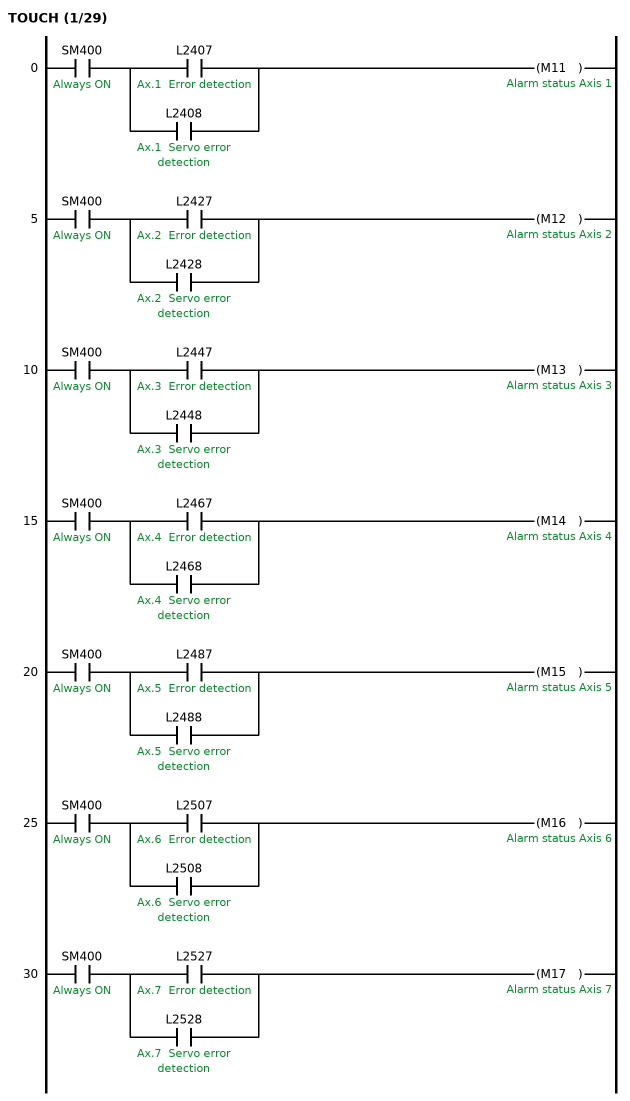
[picture p48: ladder of TOUCH, rungs at steps 0 to 30]
0     LD      SM400  ; Always ON
      LD      L2407  ; Ax.1  Error detection
      OR      L2408  ; Ax.1  Servo error detection
      ANB
      OUT     M11  ; Alarm status Axis 1
5     LD      SM400  ; Always ON
      LD      L2427  ; Ax.2  Error detection
      OR      L2428  ; Ax.2  Servo error detection
      ANB
      OUT     M12  ; Alarm status Axis 2
10    LD      SM400  ; Always ON
      LD      L2447  ; Ax.3  Error detection
      OR      L2448  ; Ax.3  Servo error detection
      ANB
      OUT     M13  ; Alarm status Axis 3
15    LD      SM400  ; Always ON
      LD      L2467  ; Ax.4  Error detection
      OR      L2468  ; Ax.4  Servo error detection
      ANB
      OUT     M14  ; Alarm status Axis 4
20    LD      SM400  ; Always ON
      LD      L2487  ; Ax.5  Error detection
      OR      L2488  ; Ax.5  Servo error detection
      ANB
      OUT     M15  ; Alarm status Axis 5
25    LD      SM400  ; Always ON
      LD      L2507  ; Ax.6  Error detection
      OR      L2508  ; Ax.6  Servo error detection
      ANB
      OUT     M16  ; Alarm status Axis 6
30    LD      SM400  ; Always ON
      LD      L2527  ; Ax.7  Error detection
      OR      L2528  ; Ax.7  Servo error detection
      ANB
      OUT     M17  ; Alarm status Axis 7
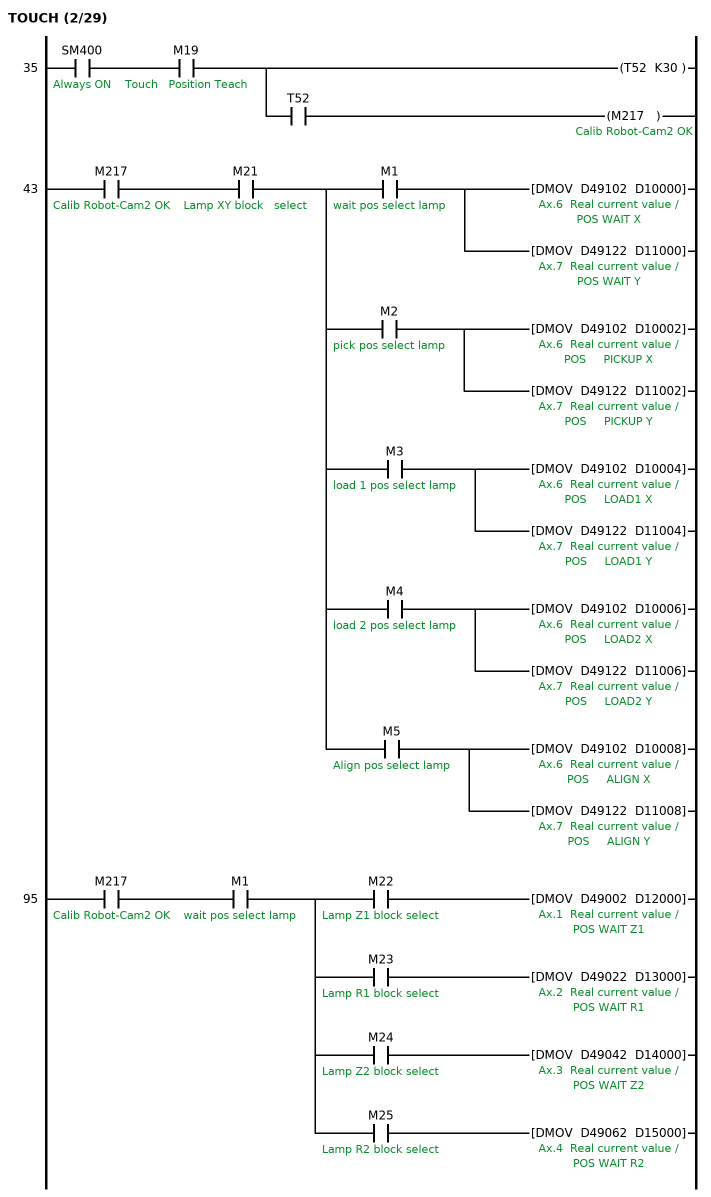
35    LD      SM400  ; Always ON
      AND     M19  ; Touch   Position Teach
      OUT     T52 K30
      AND     T52
      OUT     M217  ; Calib Robot-Cam2 OK
43    LD      M217  ; Calib Robot-Cam2 OK
      AND     M21  ; Lamp XY block   select
      MPS
      AND     M1  ; wait pos select lamp
      DMOV    D49102 D10000  ; Ax.6  Real current value / POS WAIT X
      DMOV    D49122 D11000  ; Ax.7  Real current value / POS WAIT Y
      MRD
      AND     M2  ; pick pos select lamp
      DMOV    D49102 D10002  ; POS     PICKUP X
      DMOV    D49122 D11002  ; POS     PICKUP Y
      MRD
      AND     M3  ; load 1 pos select lamp
      DMOV    D49102 D10004  ; POS     LOAD1 X
      DMOV    D49122 D11004  ; POS     LOAD1 Y
      MRD
      AND     M4  ; load 2 pos select lamp
      DMOV    D49102 D10006  ; POS     LOAD2 X
      DMOV    D49122 D11006  ; POS     LOAD2 Y
      MPP
      AND     M5  ; Align pos select lamp
      DMOV    D49102 D10008  ; POS     ALIGN X
      DMOV    D49122 D11008  ; POS     ALIGN Y
95    LD      M217  ; Calib Robot-Cam2 OK
      AND     M1  ; wait pos select lamp
      MPS
      AND     M22  ; Lamp Z1 block select
      DMOV    D49002 D12000  ; Ax.1  Real current value / POS WAIT Z1
      MRD
      AND     M23  ; Lamp R1 block select
      DMOV    D49022 D13000  ; Ax.2  Real current value / POS WAIT R1
      MRD
      AND     M24  ; Lamp Z2 block select
      DMOV    D49042 D14000  ; Ax.3  Real current value / POS WAIT Z2
      MPP
      AND     M25  ; Lamp R2 block select
      DMOV    D49062 D15000  ; Ax.4  Real current value / POS WAIT R2
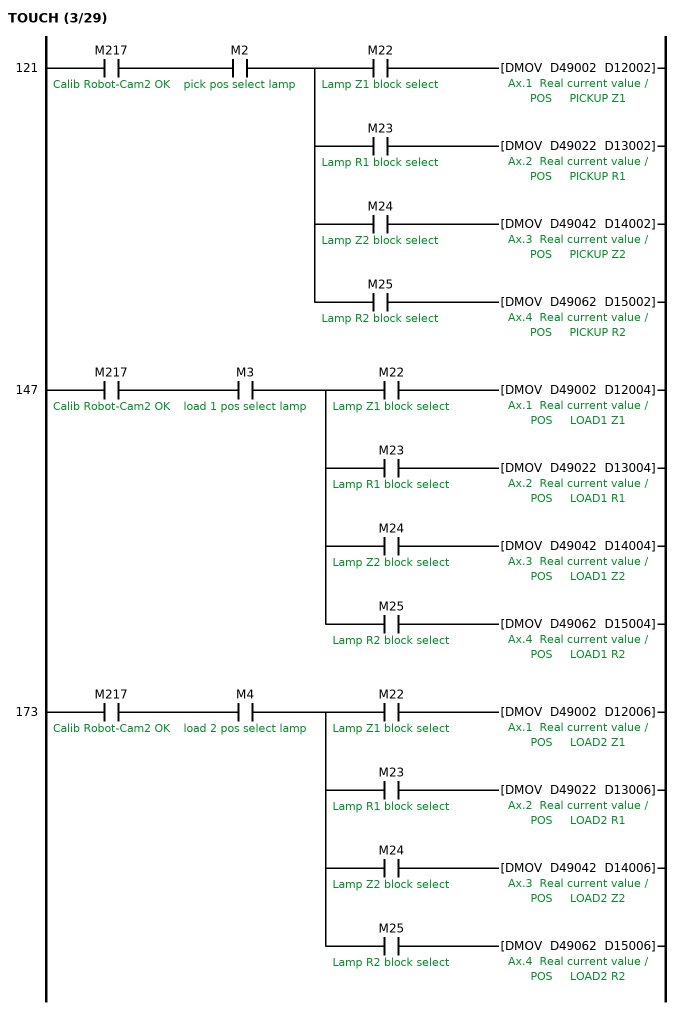
121   LD      M217  ; Calib Robot-Cam2 OK
      AND     M2  ; pick pos select lamp
      MPS
      AND     M22  ; Lamp Z1 block select
      DMOV    D49002 D12002  ; POS     PICKUP Z1
      MRD
      AND     M23  ; Lamp R1 block select
      DMOV    D49022 D13002  ; POS     PICKUP R1
      MRD
      AND     M24  ; Lamp Z2 block select
      DMOV    D49042 D14002  ; POS     PICKUP Z2
      MPP
      AND     M25  ; Lamp R2 block select
      DMOV    D49062 D15002  ; POS     PICKUP R2
147   LD      M217  ; Calib Robot-Cam2 OK
      AND     M3  ; load 1 pos select lamp
      MPS
      AND     M22  ; Lamp Z1 block select
      DMOV    D49002 D12004  ; POS     LOAD1 Z1
      MRD
      AND     M23  ; Lamp R1 block select
      DMOV    D49022 D13004  ; POS     LOAD1 R1
      MRD
      AND     M24  ; Lamp Z2 block select
      DMOV    D49042 D14004  ; POS     LOAD1 Z2
      MPP
      AND     M25  ; Lamp R2 block select
      DMOV    D49062 D15004  ; POS     LOAD1 R2
173   LD      M217  ; Calib Robot-Cam2 OK
      AND     M4  ; load 2 pos select lamp
      MPS
      AND     M22  ; Lamp Z1 block select
      DMOV    D49002 D12006  ; POS     LOAD2 Z1
      MRD
      AND     M23  ; Lamp R1 block select
      DMOV    D49022 D13006  ; POS     LOAD2 R1
      MRD
      AND     M24  ; Lamp Z2 block select
      DMOV    D49042 D14006  ; POS     LOAD2 Z2
      MPP
      AND     M25  ; Lamp R2 block select
      DMOV    D49062 D15006  ; POS     LOAD2 R2
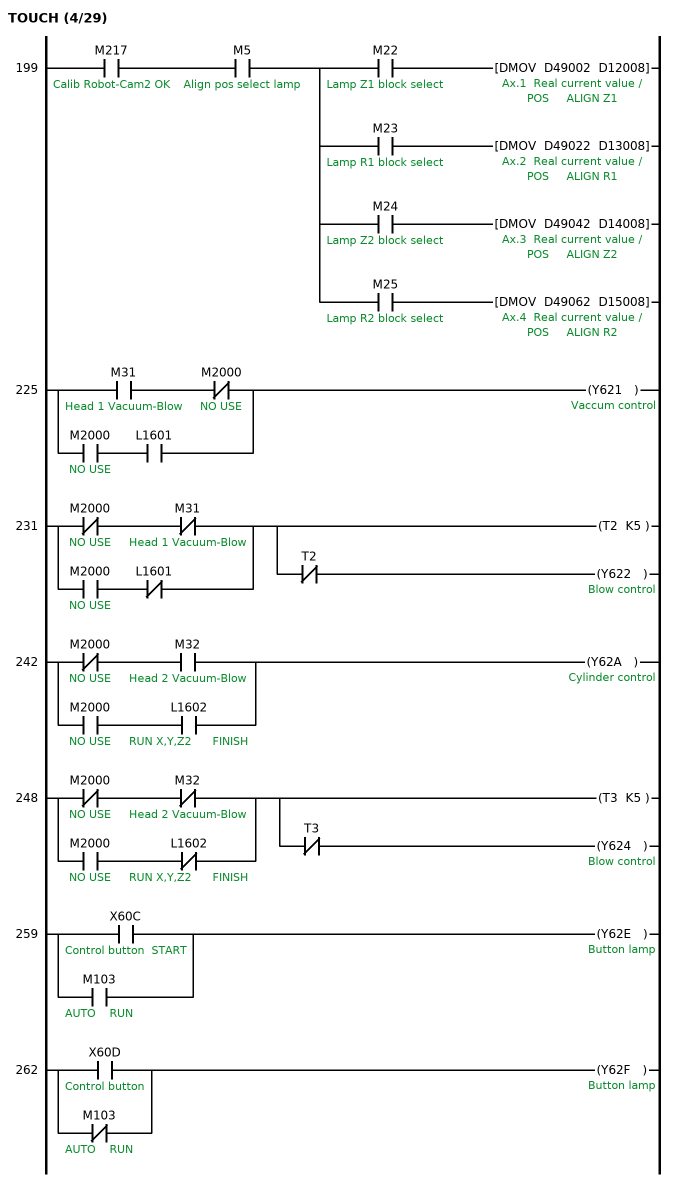
199   LD      M217  ; Calib Robot-Cam2 OK
      AND     M5  ; Align pos select lamp
      MPS
      AND     M22  ; Lamp Z1 block select
      DMOV    D49002 D12008  ; POS     ALIGN Z1
      MRD
      AND     M23  ; Lamp R1 block select
      DMOV    D49022 D13008  ; POS     ALIGN R1
      MRD
      AND     M24  ; Lamp Z2 block select
      DMOV    D49042 D14008  ; POS     ALIGN Z2
      MPP
      AND     M25  ; Lamp R2 block select
      DMOV    D49062 D15008  ; POS     ALIGN R2
225   LD      M31  ; Head 1 Vacuum-Blow
      ANI     M2000  ; NO USE
      LD      M2000  ; NO USE
      AND     L1601
      ORB
      OUT     Y621  ; Vaccum control
231   LDI     M2000  ; NO USE
      ANI     M31  ; Head 1 Vacuum-Blow
      LD      M2000  ; NO USE
      ANI     L1601
      ORB
      OUT     T2 K5
      ANI     T2
      OUT     Y622  ; Blow control
242   LDI     M2000  ; NO USE
      AND     M32  ; Head 2 Vacuum-Blow
      LD      M2000  ; NO USE
      AND     L1602  ; RUN X,Y,Z2      FINISH
      ORB
      OUT     Y62A  ; Cylinder control
248   LDI     M2000  ; NO USE
      ANI     M32  ; Head 2 Vacuum-Blow
      LD      M2000  ; NO USE
      ANI     L1602  ; RUN X,Y,Z2      FINISH
      ORB
      OUT     T3 K5
      ANI     T3
      OUT     Y624  ; Blow control
259   LD      X60C  ; Control button  START
      OR      M103  ; AUTO    RUN
      OUT     Y62E  ; Button lamp
262   LD      X60D  ; Control button
      ORI     M103  ; AUTO    RUN
      OUT     Y62F  ; Button lamp
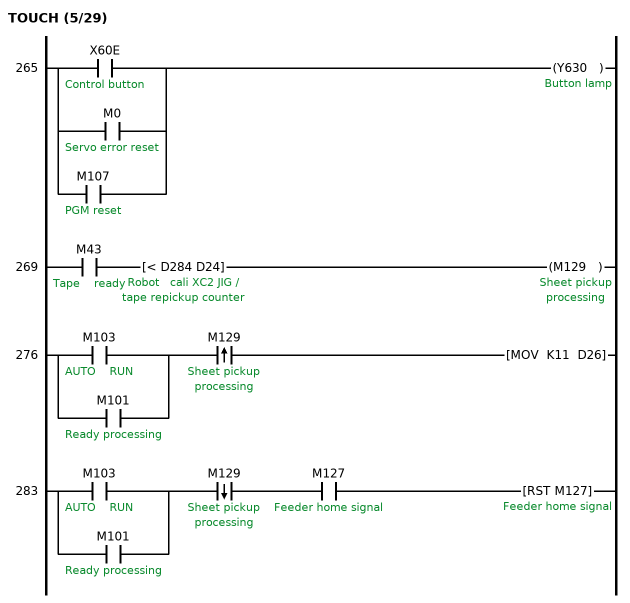
265   LD      X60E  ; Control button
      OR      M0  ; Servo error reset
      OR      M107  ; PGM reset
      OUT     Y630  ; Button lamp
269   LD      M43  ; Tape    ready
      AND<    D284 D24  ; Robot   cali XC2 JIG / tape repickup counter
      OUT     M129  ; Sheet pickup processing
276   LD      M103  ; AUTO    RUN
      OR      M101  ; Ready processing
      ANDP    M129  ; Sheet pickup processing
      MOV     K11 D26
283   LD      M103  ; AUTO    RUN
      OR      M101  ; Ready processing
      ANDF    M129  ; Sheet pickup processing
      AND     M127  ; Feeder home signal
      RST     M127  ; Feeder home signal
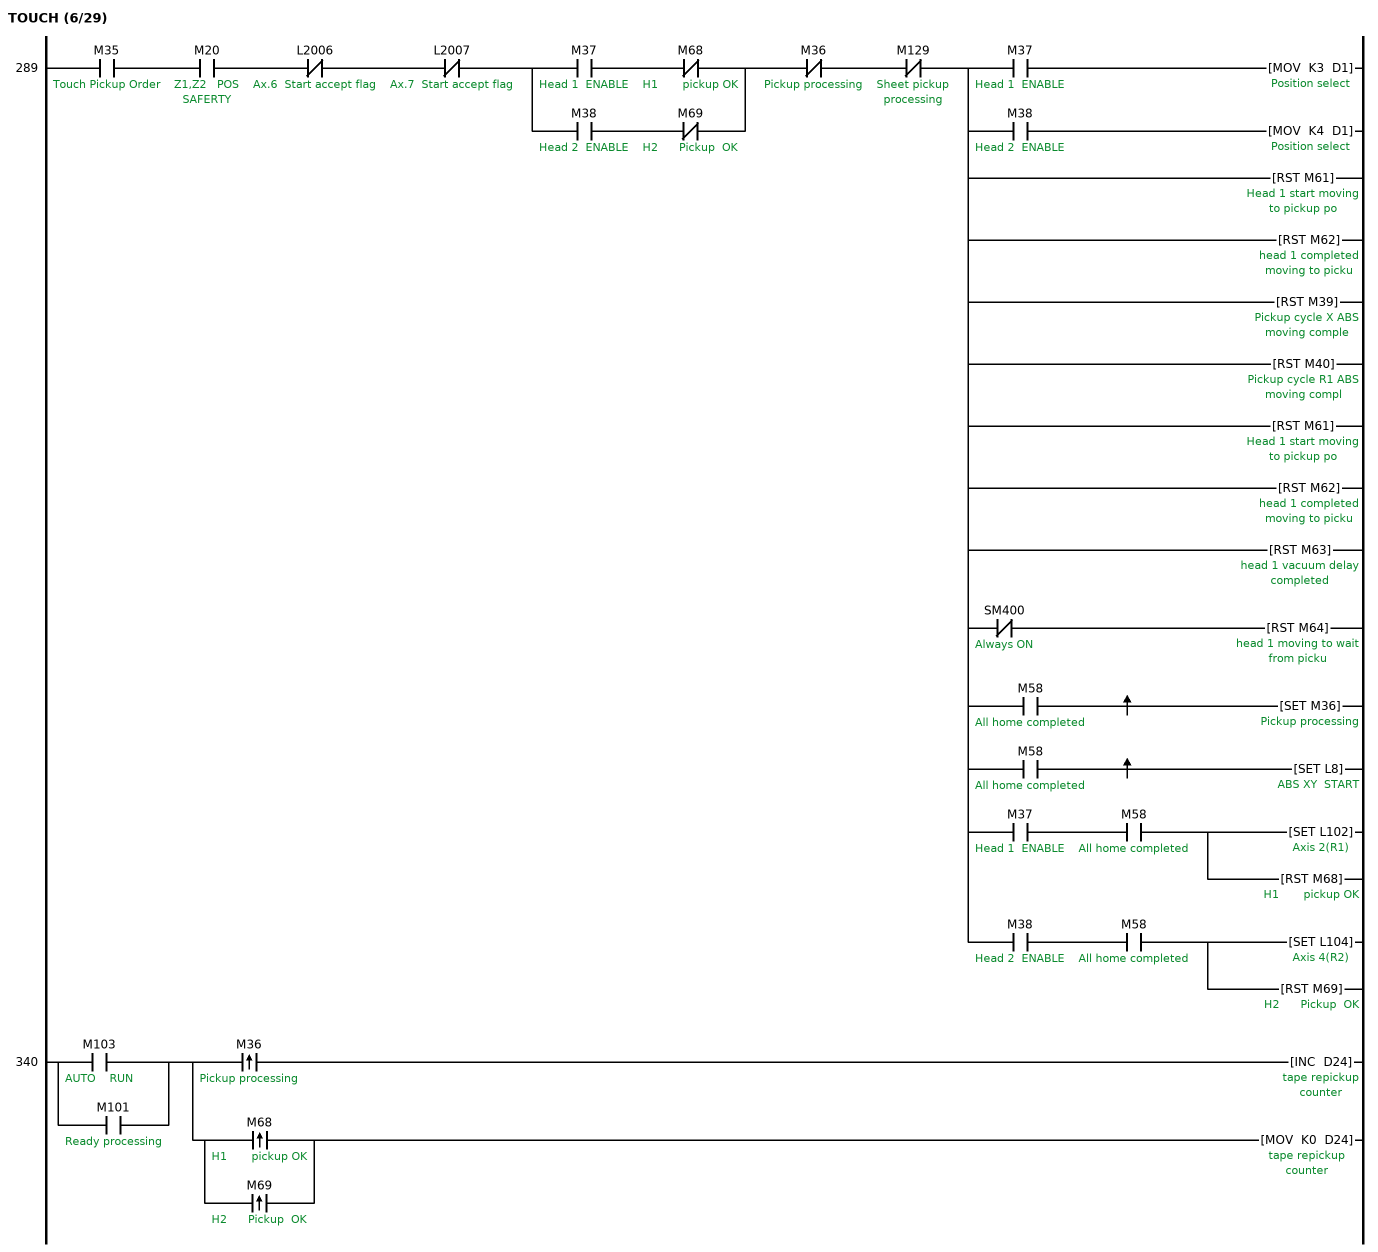
289   LD      M35  ; Touch Pickup Order
      AND     M20  ; Z1,Z2   POS     SAFERTY
      ANI     L2006  ; Ax.6  Start accept flag
      ANI     L2007  ; Ax.7  Start accept flag
      LD      M37  ; Head 1  ENABLE
      ANI     M68  ; H1       pickup OK
      LD      M38  ; Head 2  ENABLE
      ANI     M69  ; H2      Pickup  OK
      ORB
      ANB
      ANI     M36  ; Pickup processing
      ANI     M129  ; Sheet pickup processing
      MPS
      AND     M37  ; Head 1  ENABLE
      MOV     K3 D1  ; Position select
      MRD
      AND     M38  ; Head 2  ENABLE
      MOV     K4 D1
      MPP
      RST     M61  ; Head 1 start moving to pickup po
      RST     M62  ; head 1 completed moving to picku
      RST     M39  ; Pickup cycle X ABS moving comple
      RST     M40  ; Pickup cycle R1 ABS moving compl
      RST     M61  ; Head 1 start moving to pickup po
      RST     M62  ; head 1 completed moving to picku
      RST     M63  ; head 1 vacuum delay completed
      MPS
      ANI     SM400  ; Always ON
      RST     M64  ; head 1 moving to wait from picku
      MRD
      AND     M58  ; All home completed
      MEP
      SET     M36  ; Pickup processing
      MRD
      AND     M58  ; All home completed
      MEP
      SET     L8  ; ABS XY  START
      MRD
      AND     M37  ; Head 1  ENABLE
      AND     M58  ; All home completed
      SET     L102  ; Axis 2(R1)
      RST     M68  ; H1       pickup OK
      MPP
      AND     M38  ; Head 2  ENABLE
      AND     M58  ; All home completed
      SET     L104  ; Axis 4(R2)
      RST     M69  ; H2      Pickup  OK
340   LD      M103  ; AUTO    RUN
      OR      M101  ; Ready processing
      MPS
      ANDP    M36  ; Pickup processing
      INC     D24
      MPP
      LDP     M68  ; H1       pickup OK
      ORP     M69  ; H2      Pickup  OK
      ANB
      MOV     K0 D24
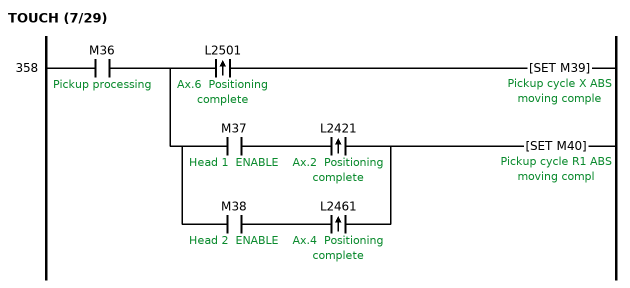
358   LD      M36  ; Pickup processing
      MPS
      ANDP    L2501  ; Ax.6  Positioning complete
      SET     M39  ; Pickup cycle X ABS moving comple
      MPP
      LD      M37  ; Head 1  ENABLE
      ANDP    L2421  ; Ax.2  Positioning complete
      LD      M38  ; Head 2  ENABLE
      ANDP    L2461  ; Ax.4  Positioning complete
      ORB
      ANB
      SET     M40  ; Pickup cycle R1 ABS moving compl
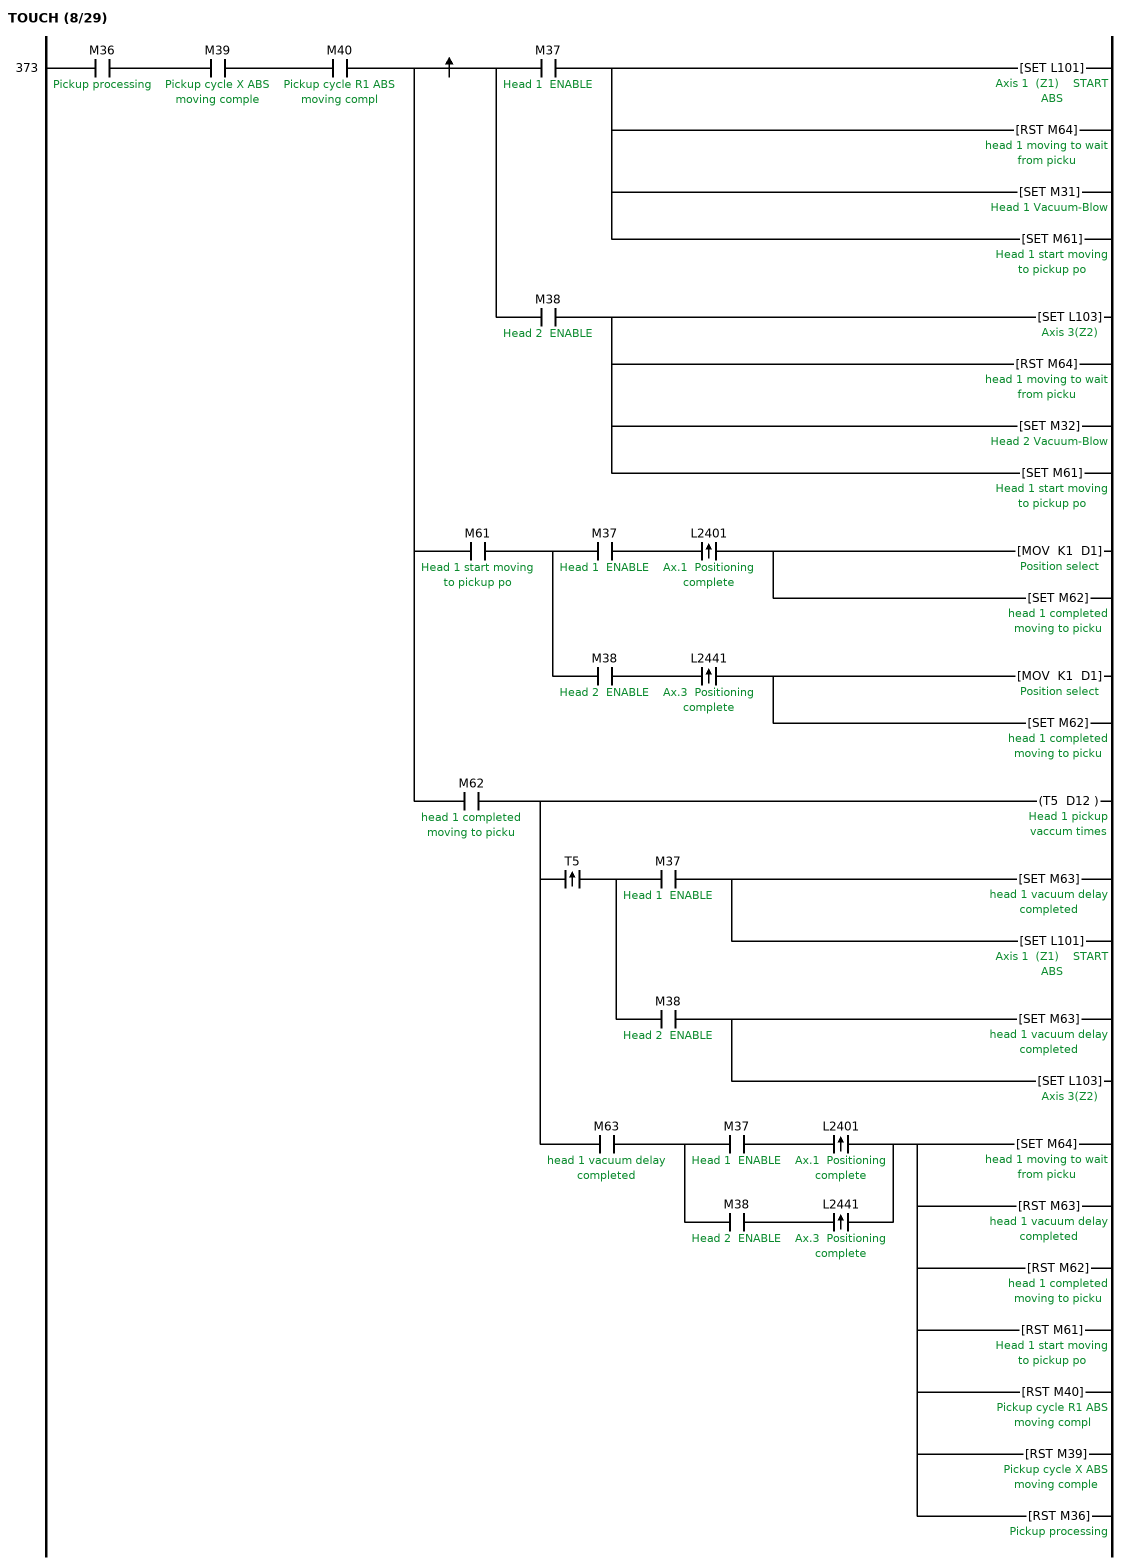
373   LD      M36  ; Pickup processing
      AND     M39  ; Pickup cycle X ABS moving comple
      AND     M40  ; Pickup cycle R1 ABS moving compl
      MPS
      MEP
      MPS
      AND     M37  ; Head 1  ENABLE
      SET     L101  ; Axis 1  (Z1)    START   ABS
      RST     M64  ; head 1 moving to wait from picku
      SET     M31  ; Head 1 Vacuum-Blow
      SET     M61  ; Head 1 start moving to pickup po
      MPP
      AND     M38  ; Head 2  ENABLE
      SET     L103  ; Axis 3(Z2)
      RST     M64  ; head 1 moving to wait from picku
      SET     M32  ; Head 2 Vacuum-Blow
      SET     M61  ; Head 1 start moving to pickup po
      MRD
      AND     M61  ; Head 1 start moving to pickup po
      MPS
      AND     M37  ; Head 1  ENABLE
      ANDP    L2401  ; Ax.1  Positioning complete
      MOV     K1 D1
      SET     M62  ; head 1 completed moving to picku
      MPP
      AND     M38  ; Head 2  ENABLE
      ANDP    L2441  ; Ax.3  Positioning complete
      MOV     K1 D1
      SET     M62  ; head 1 completed moving to picku
      MPP
      AND     M62  ; head 1 completed moving to picku
      OUT     T5 D12  ; Head 1 pickup vaccum times
      MPS
      ANDP    T5
      MPS
      AND     M37  ; Head 1  ENABLE
      SET     M63  ; head 1 vacuum delay completed
      SET     L101  ; Axis 1  (Z1)    START   ABS
      MPP
      AND     M38  ; Head 2  ENABLE
      SET     M63  ; head 1 vacuum delay completed
      SET     L103  ; Axis 3(Z2)
      MPP
      AND     M63  ; head 1 vacuum delay completed
      LD      M37  ; Head 1  ENABLE
      ANDP    L2401  ; Ax.1  Positioning complete
      LD      M38  ; Head 2  ENABLE
      ANDP    L2441  ; Ax.3  Positioning complete
      ORB
      ANB
      SET     M64  ; head 1 moving to wait from picku
      RST     M63  ; head 1 vacuum delay completed
      RST     M62  ; head 1 completed moving to picku
      RST     M61  ; Head 1 start moving to pickup po
      RST     M40  ; Pickup cycle R1 ABS moving compl
      RST     M39  ; Pickup cycle X ABS moving comple
      RST     M36  ; Pickup processing
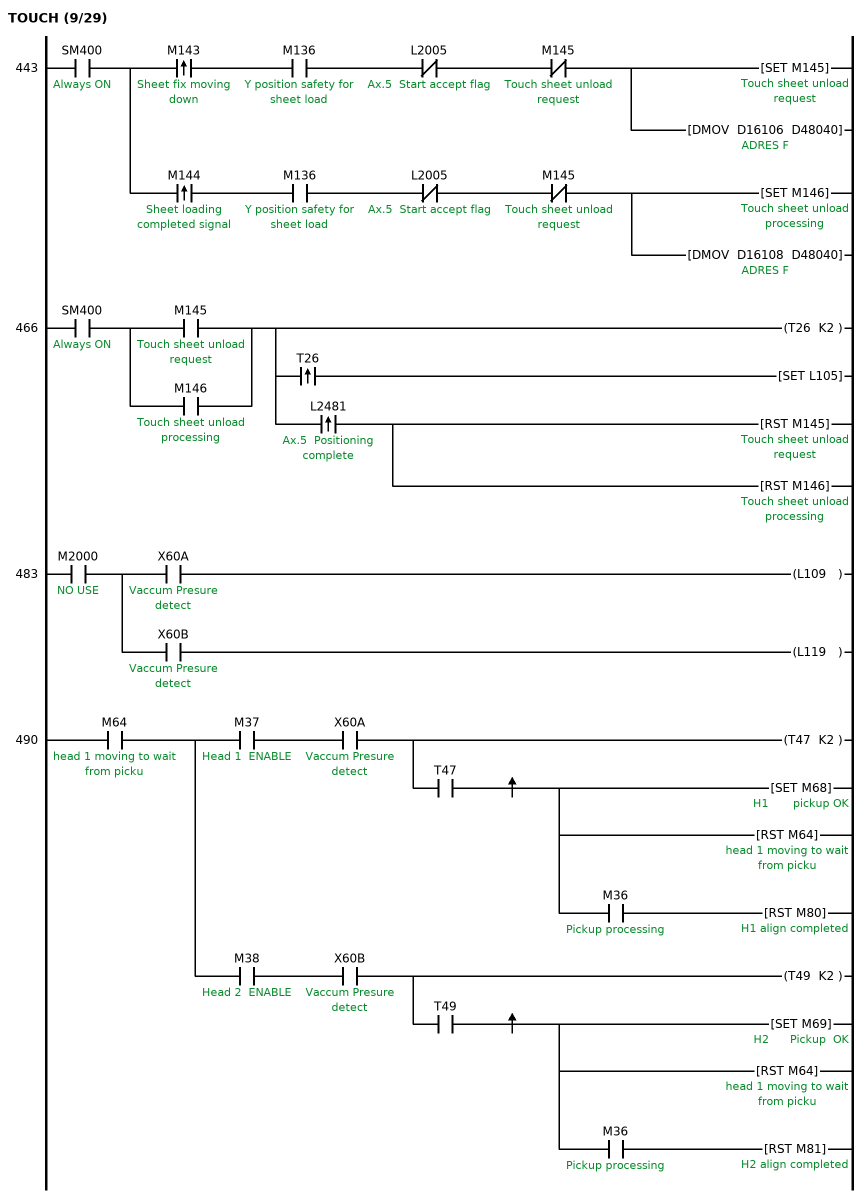
443   LD      SM400  ; Always ON
      MPS
      ANDP    M143  ; Sheet fix moving down
      AND     M136  ; Y position safety for sheet load
      ANI     L2005  ; Ax.5  Start accept flag
      ANI     M145  ; Touch sheet unload request
      SET     M145  ; Touch sheet unload request
      DMOV    D16106 D48040  ; ADRES F
      MPP
      ANDP    M144  ; Sheet loading completed signal
      AND     M136  ; Y position safety for sheet load
      ANI     L2005  ; Ax.5  Start accept flag
      ANI     M145  ; Touch sheet unload request
      SET     M146  ; Touch sheet unload processing
      DMOV    D16108 D48040
466   LD      SM400  ; Always ON
      LD      M145  ; Touch sheet unload request
      OR      M146  ; Touch sheet unload processing
      ANB
      OUT     T26 K2
      MPS
      ANDP    T26
      SET     L105
      MPP
      ANDP    L2481  ; Ax.5  Positioning complete
      RST     M145  ; Touch sheet unload request
      RST     M146  ; Touch sheet unload processing
483   LD      M2000  ; NO USE
      MPS
      AND     X60A  ; Vaccum Presure detect
      OUT     L109
      MPP
      AND     X60B  ; Vaccum Presure detect
      OUT     L119
490   LD      M64  ; head 1 moving to wait from picku
      MPS
      AND     M37  ; Head 1  ENABLE
      AND     X60A  ; Vaccum Presure detect
      OUT     T47 K2
      AND     T47
      MEP
      SET     M68  ; H1       pickup OK
      RST     M64  ; head 1 moving to wait from picku
      AND     M36  ; Pickup processing
      RST     M80  ; H1 align completed
      MPP
      AND     M38  ; Head 2  ENABLE
      AND     X60B  ; Vaccum Presure detect
      OUT     T49 K2
      AND     T49
      MEP
      SET     M69  ; H2      Pickup  OK
      RST     M64  ; head 1 moving to wait from picku
      AND     M36  ; Pickup processing
      RST     M81  ; H2 align completed
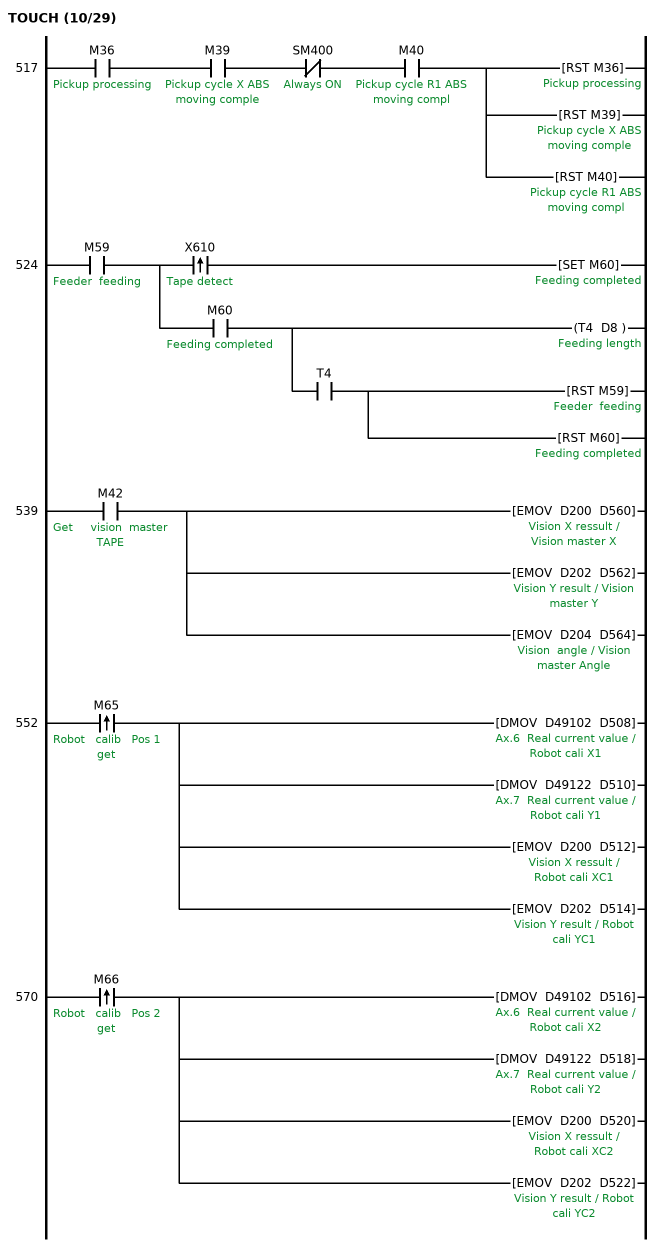
517   LD      M36  ; Pickup processing
      AND     M39  ; Pickup cycle X ABS moving comple
      ANI     SM400  ; Always ON
      AND     M40  ; Pickup cycle R1 ABS moving compl
      RST     M36  ; Pickup processing
      RST     M39  ; Pickup cycle X ABS moving comple
      RST     M40  ; Pickup cycle R1 ABS moving compl
524   LD      M59  ; Feeder  feeding
      MPS
      ANDP    X610  ; Tape detect
      SET     M60  ; Feeding completed
      MPP
      AND     M60  ; Feeding completed
      OUT     T4 D8  ; Feeding length
      AND     T4
      RST     M59  ; Feeder  feeding
      RST     M60  ; Feeding completed
539   LD      M42  ; Get     vision  master  TAPE
      EMOV    D200 D560  ; Vision X ressult / Vision master X
      EMOV    D202 D562  ; Vision Y result / Vision master Y
      EMOV    D204 D564  ; Vision  angle / Vision master Angle
552   LDP     M65  ; Robot   calib   Pos 1   get
      DMOV    D49102 D508  ; Robot cali X1
      DMOV    D49122 D510  ; Robot cali Y1
      EMOV    D200 D512  ; Robot cali XC1
      EMOV    D202 D514  ; Robot cali YC1
570   LDP     M66  ; Robot   calib   Pos 2   get
      DMOV    D49102 D516  ; Robot cali X2
      DMOV    D49122 D518  ; Robot cali Y2
      EMOV    D200 D520  ; Robot cali XC2
      EMOV    D202 D522  ; Robot cali YC2
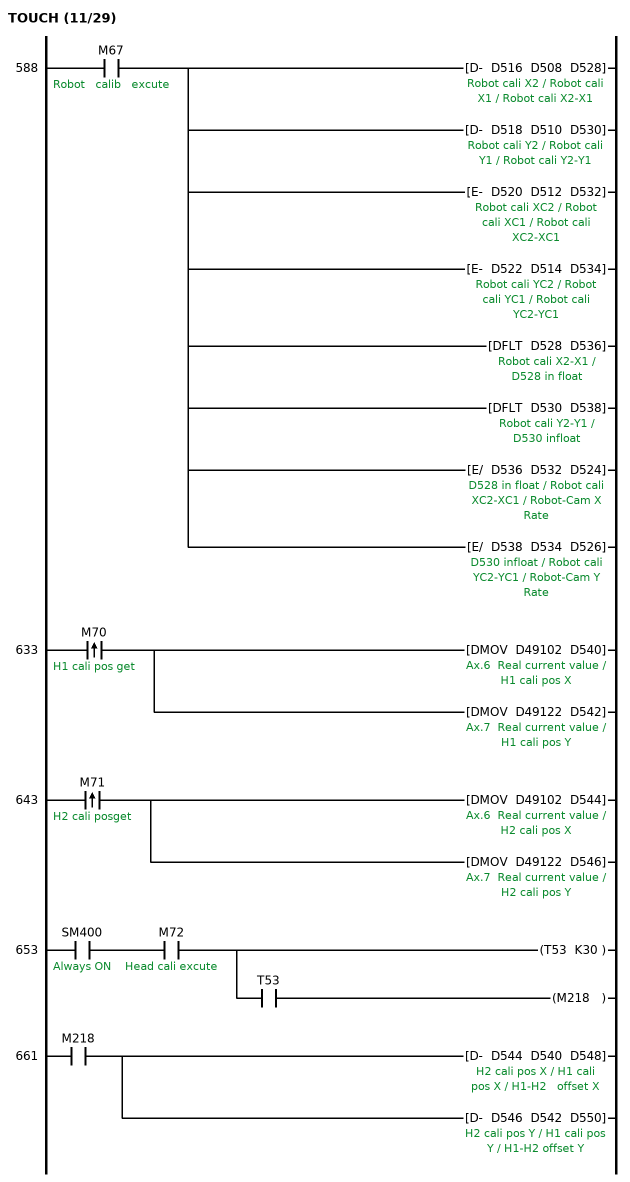
588   LD      M67  ; Robot   calib   excute
      D-      D516 D508 D528  ; Robot cali X2-X1
      D-      D518 D510 D530  ; Robot cali Y2-Y1
      E-      D520 D512 D532  ; Robot cali XC2-XC1
      E-      D522 D514 D534  ; Robot cali YC2-YC1
      DFLT    D528 D536  ; D528 in float
      DFLT    D530 D538  ; D530 infloat
      E/      D536 D532 D524  ; Robot-Cam X Rate
      E/      D538 D534 D526  ; Robot-Cam Y Rate
633   LDP     M70  ; H1 cali pos get
      DMOV    D49102 D540  ; H1 cali pos X
      DMOV    D49122 D542  ; H1 cali pos Y
643   LDP     M71  ; H2 cali posget
      DMOV    D49102 D544  ; H2 cali pos X
      DMOV    D49122 D546  ; H2 cali pos Y
653   LD      SM400  ; Always ON
      AND     M72  ; Head cali excute
      OUT     T53 K30
      AND     T53
      OUT     M218
661   LD      M218
      D-      D544 D540 D548  ; H1-H2   offset X
      D-      D546 D542 D550  ; H1-H2 offset Y
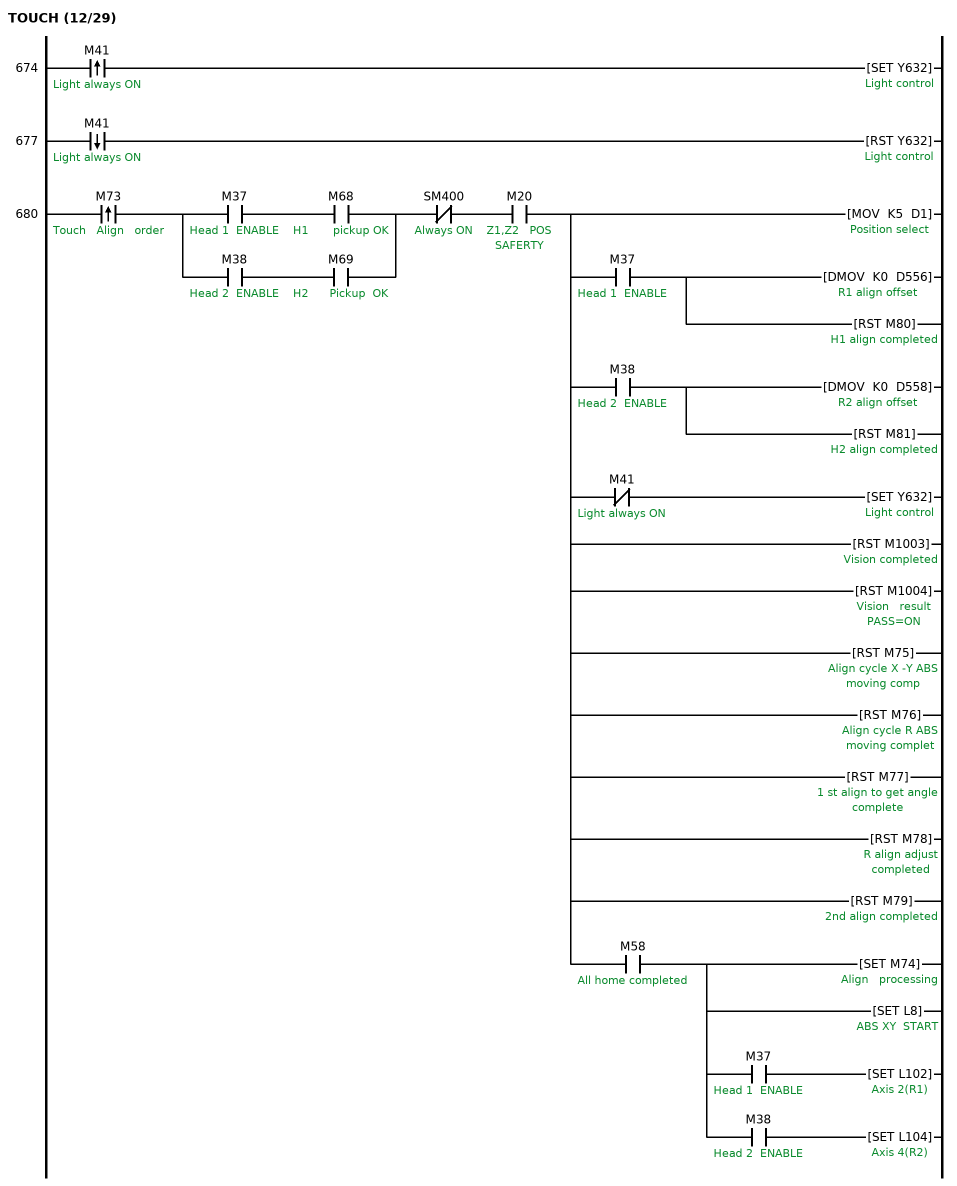
674   LDP     M41  ; Light always ON
      SET     Y632  ; Light control
677   LDF     M41  ; Light always ON
      RST     Y632  ; Light control
680   LDP     M73  ; Touch   Align   order
      LD      M37  ; Head 1  ENABLE
      AND     M68  ; H1       pickup OK
      LD      M38  ; Head 2  ENABLE
      AND     M69  ; H2      Pickup  OK
      ORB
      ANB
      ANI     SM400  ; Always ON
      AND     M20  ; Z1,Z2   POS     SAFERTY
      MOV     K5 D1
      MPS
      AND     M37  ; Head 1  ENABLE
      DMOV    K0 D556  ; R1 align offset
      RST     M80  ; H1 align completed
      MRD
      AND     M38  ; Head 2  ENABLE
      DMOV    K0 D558  ; R2 align offset
      RST     M81  ; H2 align completed
      MRD
      ANI     M41  ; Light always ON
      SET     Y632  ; Light control
      MPP
      RST     M1003  ; Vision completed
      RST     M1004  ; Vision   result PASS=ON
      RST     M75  ; Align cycle X -Y ABS moving comp
      RST     M76  ; Align cycle R ABS moving complet
      RST     M77  ; 1 st align to get angle complete
      RST     M78  ; R align adjust completed
      RST     M79  ; 2nd align completed
      AND     M58  ; All home completed
      SET     M74  ; Align   processing
      SET     L8  ; ABS XY  START
      MPS
      AND     M37  ; Head 1  ENABLE
      SET     L102  ; Axis 2(R1)
      MPP
      AND     M38  ; Head 2  ENABLE
      SET     L104  ; Axis 4(R2)
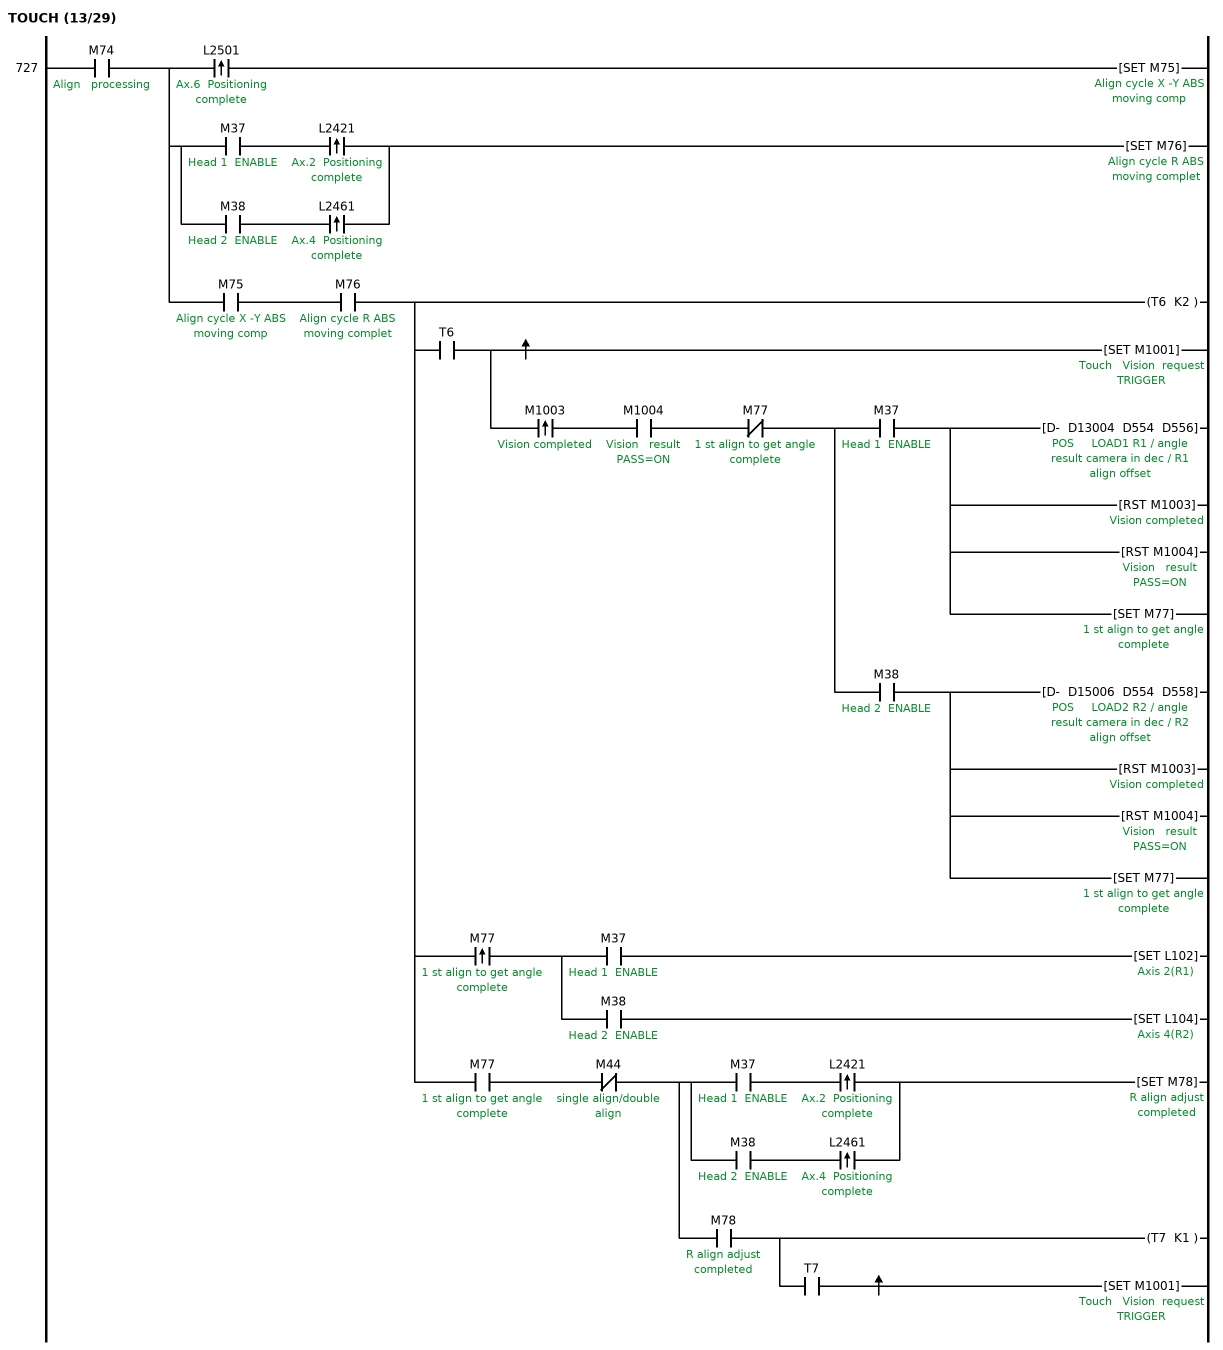
727   LD      M74  ; Align   processing
      MPS
      ANDP    L2501  ; Ax.6  Positioning complete
      SET     M75  ; Align cycle X -Y ABS moving comp
      MRD
      LD      M37  ; Head 1  ENABLE
      ANDP    L2421  ; Ax.2  Positioning complete
      LD      M38  ; Head 2  ENABLE
      ANDP    L2461  ; Ax.4  Positioning complete
      ORB
      ANB
      SET     M76  ; Align cycle R ABS moving complet
      MPP
      AND     M75  ; Align cycle X -Y ABS moving comp
      AND     M76  ; Align cycle R ABS moving complet
      OUT     T6 K2
      MPS
      AND     T6
      MPS
      MEP
      SET     M1001  ; Touch   Vision  request TRIGGER
      MPP
      ANDP    M1003  ; Vision completed
      AND     M1004  ; Vision   result PASS=ON
      ANI     M77  ; 1 st align to get angle complete
      MPS
      AND     M37  ; Head 1  ENABLE
      D-      D13004 D554 D556  ; angle result camera in dec
      RST     M1003  ; Vision completed
      RST     M1004  ; Vision   result PASS=ON
      SET     M77  ; 1 st align to get angle complete
      MPP
      AND     M38  ; Head 2  ENABLE
      D-      D15006 D554 D558
      RST     M1003  ; Vision completed
      RST     M1004  ; Vision   result PASS=ON
      SET     M77  ; 1 st align to get angle complete
      MRD
      ANDP    M77  ; 1 st align to get angle complete
      MPS
      AND     M37  ; Head 1  ENABLE
      SET     L102  ; Axis 2(R1)
      MPP
      AND     M38  ; Head 2  ENABLE
      SET     L104  ; Axis 4(R2)
      MPP
      AND     M77  ; 1 st align to get angle complete
      ANI     M44  ; single align/double align
      MPS
      LD      M37  ; Head 1  ENABLE
      ANDP    L2421  ; Ax.2  Positioning complete
      LD      M38  ; Head 2  ENABLE
      ANDP    L2461  ; Ax.4  Positioning complete
      ORB
      ANB
      SET     M78  ; R align adjust completed
      MPP
      AND     M78  ; R align adjust completed
      OUT     T7 K1
      AND     T7
      MEP
      SET     M1001  ; Touch   Vision  request TRIGGER
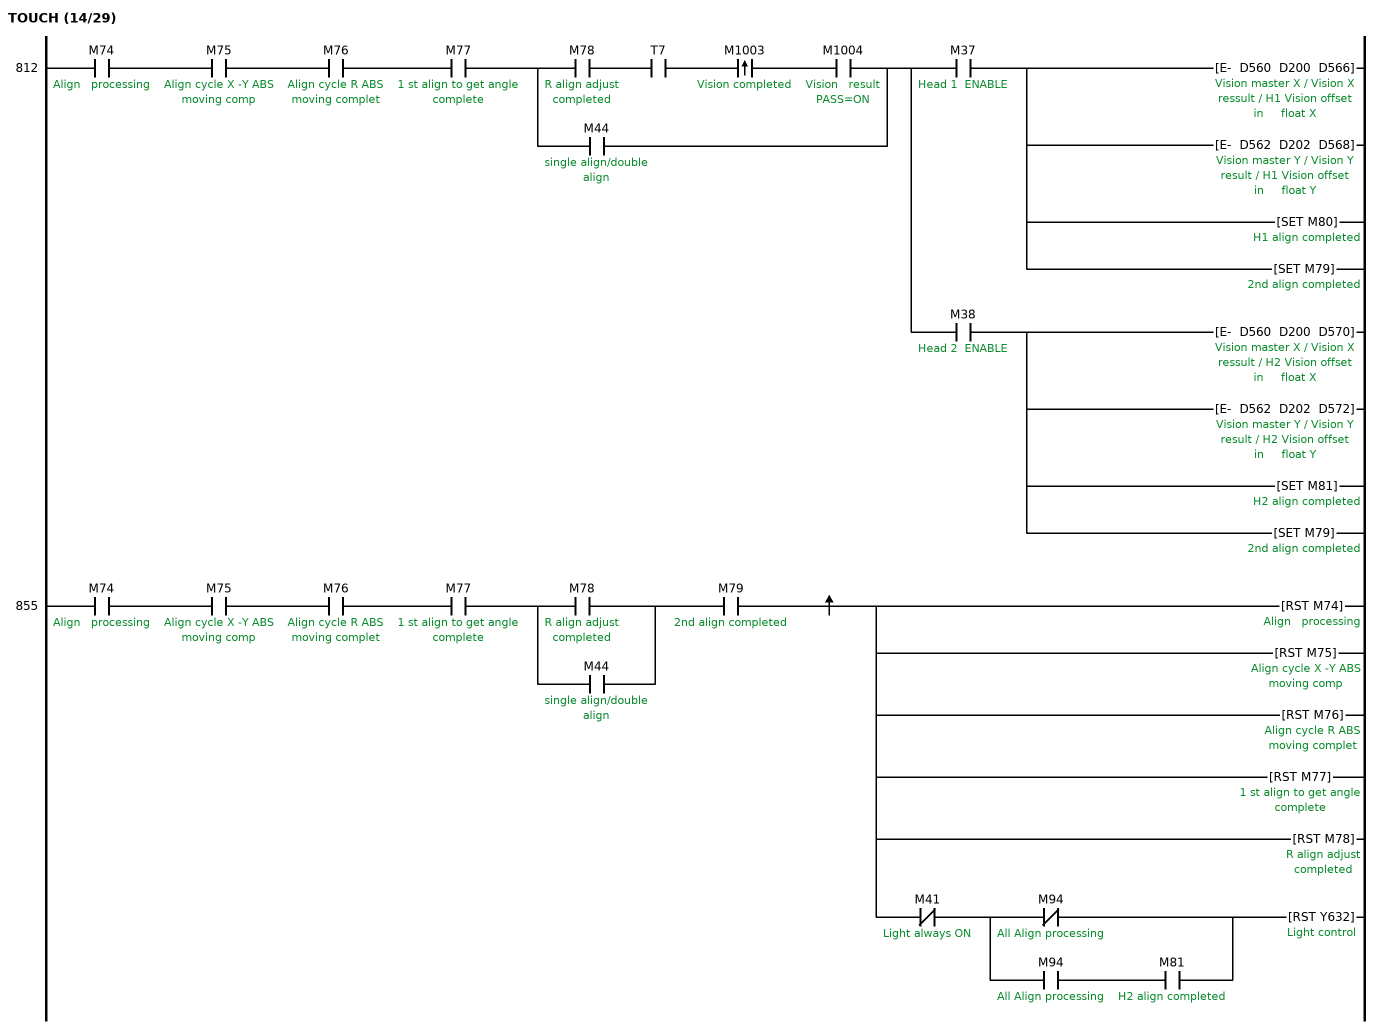
812   LD      M74  ; Align   processing
      AND     M75  ; Align cycle X -Y ABS moving comp
      AND     M76  ; Align cycle R ABS moving complet
      AND     M77  ; 1 st align to get angle complete
      LD      M78  ; R align adjust completed
      AND     T7
      ANDP    M1003  ; Vision completed
      AND     M1004  ; Vision   result PASS=ON
      OR      M44  ; single align/double align
      ANB
      MPS
      AND     M37  ; Head 1  ENABLE
      E-      D560 D200 D566  ; H1 Vision offset in     float X
      E-      D562 D202 D568  ; H1 Vision offset in     float Y
      SET     M80  ; H1 align completed
      SET     M79  ; 2nd align completed
      MPP
      AND     M38  ; Head 2  ENABLE
      E-      D560 D200 D570  ; H2 Vision offset in     float X
      E-      D562 D202 D572  ; H2 Vision offset in     float Y
      SET     M81  ; H2 align completed
      SET     M79  ; 2nd align completed
855   LD      M74  ; Align   processing
      AND     M75  ; Align cycle X -Y ABS moving comp
      AND     M76  ; Align cycle R ABS moving complet
      AND     M77  ; 1 st align to get angle complete
      LD      M78  ; R align adjust completed
      OR      M44  ; single align/double align
      ANB
      AND     M79  ; 2nd align completed
      MEP
      RST     M74  ; Align   processing
      RST     M75  ; Align cycle X -Y ABS moving comp
      RST     M76  ; Align cycle R ABS moving complet
      RST     M77  ; 1 st align to get angle complete
      RST     M78  ; R align adjust completed
      ANI     M41  ; Light always ON
      LDI     M94  ; All Align processing
      LD      M94  ; All Align processing
      AND     M81  ; H2 align completed
      ORB
      ANB
      RST     Y632  ; Light control
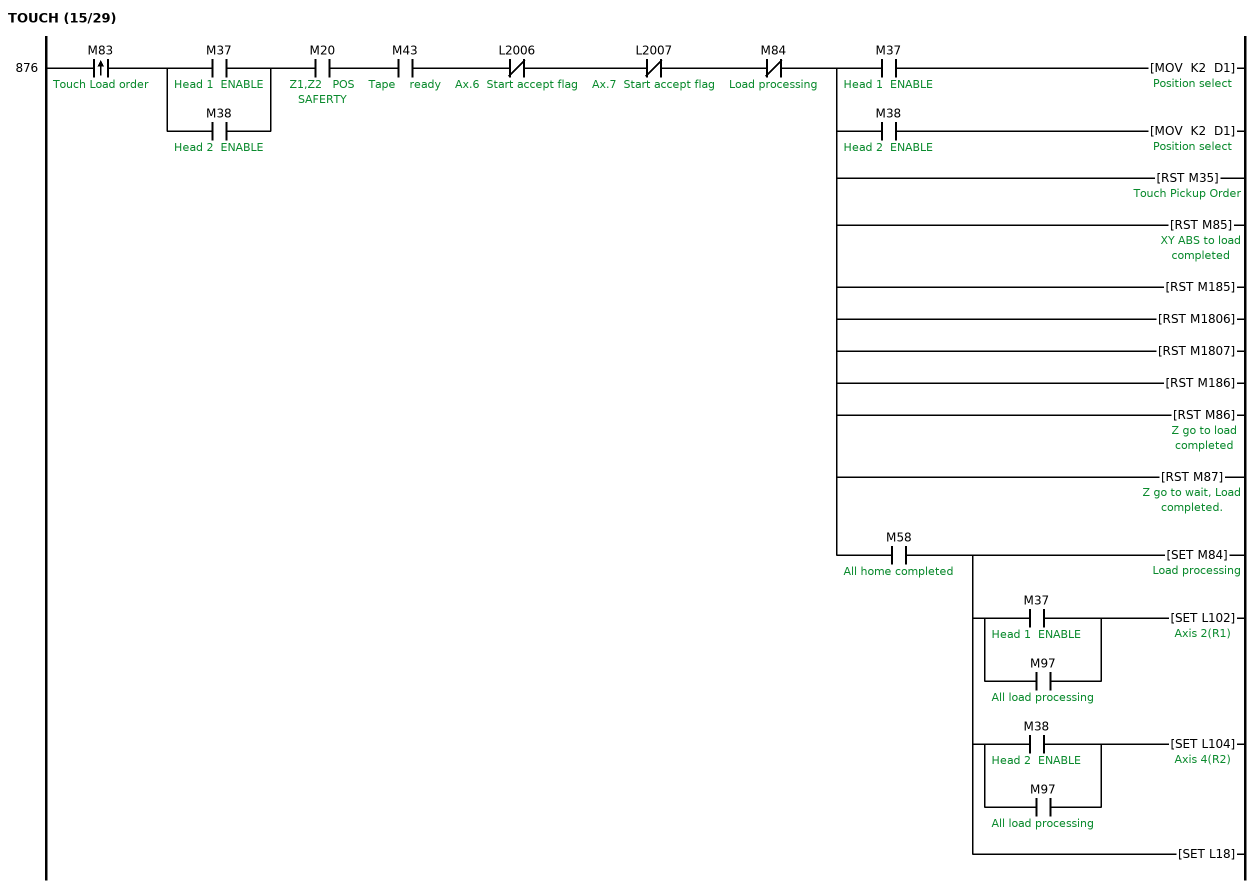
876   LDP     M83  ; Touch Load order
      LD      M37  ; Head 1  ENABLE
      OR      M38  ; Head 2  ENABLE
      ANB
      AND     M20  ; Z1,Z2   POS     SAFERTY
      AND     M43  ; Tape    ready
      ANI     L2006  ; Ax.6  Start accept flag
      ANI     L2007  ; Ax.7  Start accept flag
      ANI     M84  ; Load processing
      MPS
      AND     M37  ; Head 1  ENABLE
      MOV     K2 D1
      MRD
      AND     M38  ; Head 2  ENABLE
      MOV     K2 D1
      MPP
      RST     M35  ; Touch Pickup Order
      RST     M85  ; XY ABS to load completed
      RST     M185
      RST     M1806
      RST     M1807
      RST     M186
      RST     M86  ; Z go to load completed
      RST     M87  ; Z go to wait, Load completed.
      AND     M58  ; All home completed
      SET     M84  ; Load processing
      MPS
      LD      M37  ; Head 1  ENABLE
      OR      M97  ; All load processing
      ANB
      SET     L102  ; Axis 2(R1)
      MRD
      LD      M38  ; Head 2  ENABLE
      OR      M97  ; All load processing
      ANB
      SET     L104  ; Axis 4(R2)
      MPP
      SET     L18
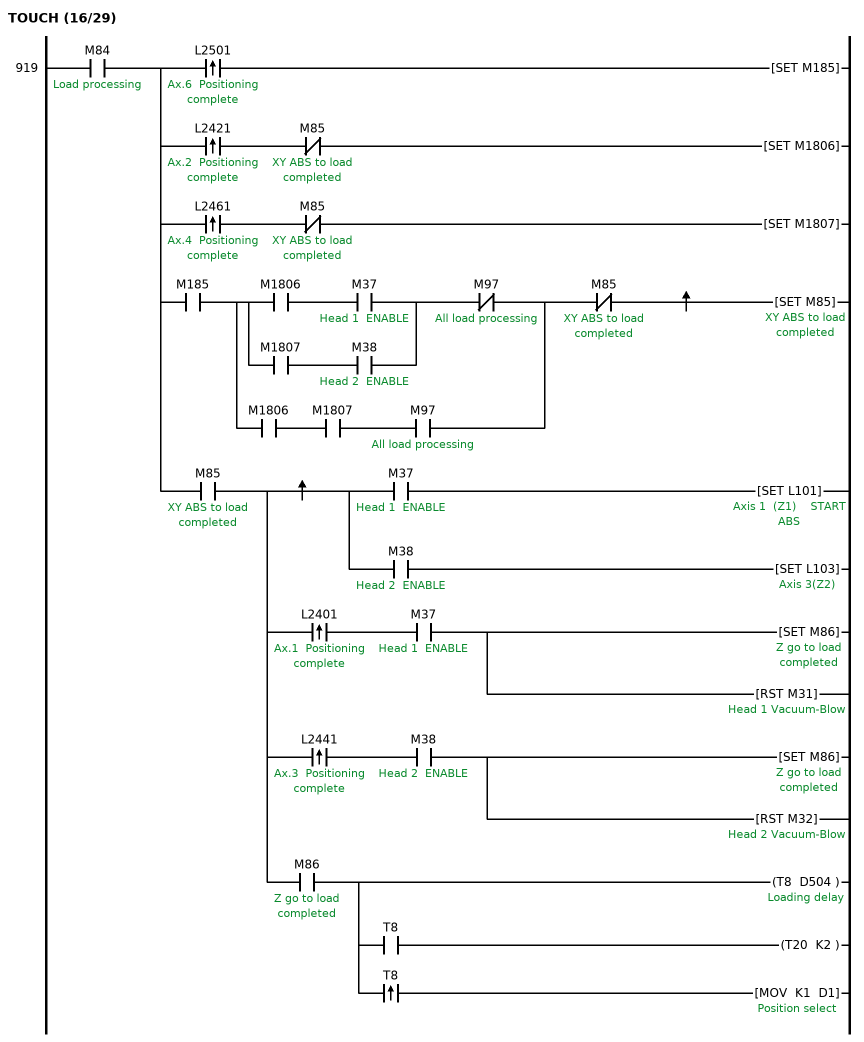
919   LD      M84  ; Load processing
      MPS
      ANDP    L2501  ; Ax.6  Positioning complete
      SET     M185
      MRD
      ANDP    L2421  ; Ax.2  Positioning complete
      ANI     M85  ; XY ABS to load completed
      SET     M1806
      MRD
      ANDP    L2461  ; Ax.4  Positioning complete
      ANI     M85  ; XY ABS to load completed
      SET     M1807
      MRD
      AND     M185
      LD      M1806
      AND     M37  ; Head 1  ENABLE
      LD      M1807
      AND     M38  ; Head 2  ENABLE
      ORB
      ANI     M97  ; All load processing
      LD      M1806
      AND     M1807
      AND     M97  ; All load processing
      ORB
      ANB
      ANI     M85  ; XY ABS to load completed
      MEP
      SET     M85  ; XY ABS to load completed
      MPP
      AND     M85  ; XY ABS to load completed
      MPS
      MEP
      MPS
      AND     M37  ; Head 1  ENABLE
      SET     L101  ; Axis 1  (Z1)    START   ABS
      MPP
      AND     M38  ; Head 2  ENABLE
      SET     L103  ; Axis 3(Z2)
      MRD
      ANDP    L2401  ; Ax.1  Positioning complete
      AND     M37  ; Head 1  ENABLE
      SET     M86  ; Z go to load completed
      RST     M31  ; Head 1 Vacuum-Blow
      MRD
      ANDP    L2441  ; Ax.3  Positioning complete
      AND     M38  ; Head 2  ENABLE
      SET     M86  ; Z go to load completed
      RST     M32  ; Head 2 Vacuum-Blow
      MPP
      AND     M86  ; Z go to load completed
      OUT     T8 D504  ; Loading delay
      MPS
      AND     T8
      OUT     T20 K2
      MPP
      ANDP    T8
      MOV     K1 D1
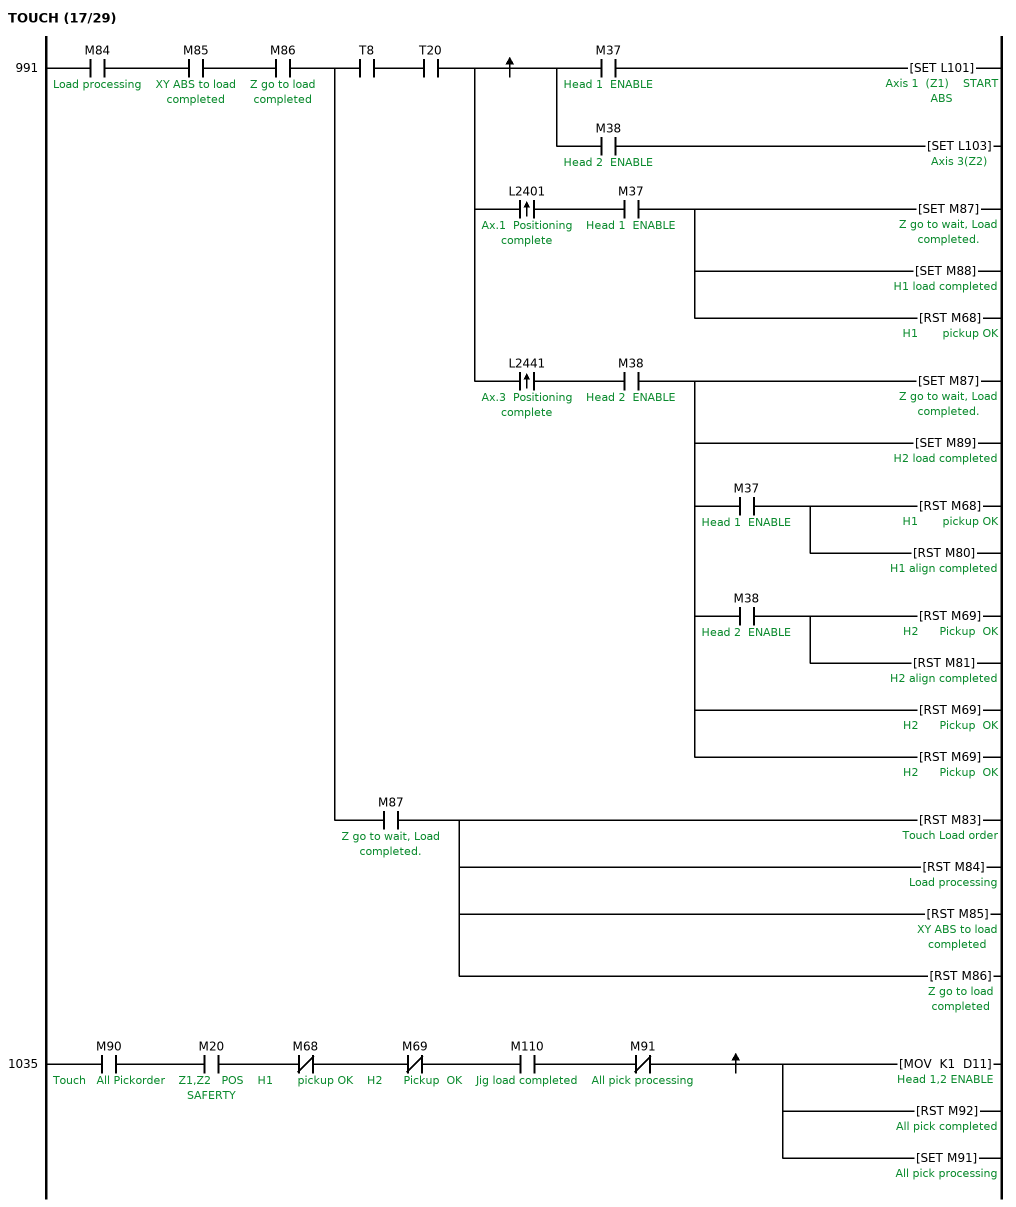
991   LD      M84  ; Load processing
      AND     M85  ; XY ABS to load completed
      AND     M86  ; Z go to load completed
      MPS
      AND     T8
      AND     T20
      MPS
      MEP
      MPS
      AND     M37  ; Head 1  ENABLE
      SET     L101  ; Axis 1  (Z1)    START   ABS
      MPP
      AND     M38  ; Head 2  ENABLE
      SET     L103  ; Axis 3(Z2)
      MRD
      ANDP    L2401  ; Ax.1  Positioning complete
      AND     M37  ; Head 1  ENABLE
      SET     M87  ; Z go to wait, Load completed.
      SET     M88  ; H1 load completed
      RST     M68  ; H1       pickup OK
      MPP
      ANDP    L2441  ; Ax.3  Positioning complete
      AND     M38  ; Head 2  ENABLE
      SET     M87  ; Z go to wait, Load completed.
      SET     M89  ; H2 load completed
      MPS
      AND     M37  ; Head 1  ENABLE
      RST     M68  ; H1       pickup OK
      RST     M80  ; H1 align completed
      MRD
      AND     M38  ; Head 2  ENABLE
      RST     M69  ; H2      Pickup  OK
      RST     M81  ; H2 align completed
      MPP
      RST     M69  ; H2      Pickup  OK
      RST     M69  ; H2      Pickup  OK
      MPP
      AND     M87  ; Z go to wait, Load completed.
      RST     M83  ; Touch Load order
      RST     M84  ; Load processing
      RST     M85  ; XY ABS to load completed
      RST     M86  ; Z go to load completed
1035  LD      M90  ; Touch   All Pickorder
      AND     M20  ; Z1,Z2   POS     SAFERTY
      ANI     M68  ; H1       pickup OK
      ANI     M69  ; H2      Pickup  OK
      AND     M110  ; Jig load completed
      ANI     M91  ; All pick processing
      MEP
      MOV     K1 D11  ; Head 1,2 ENABLE
      RST     M92  ; All pick completed
      SET     M91  ; All pick processing
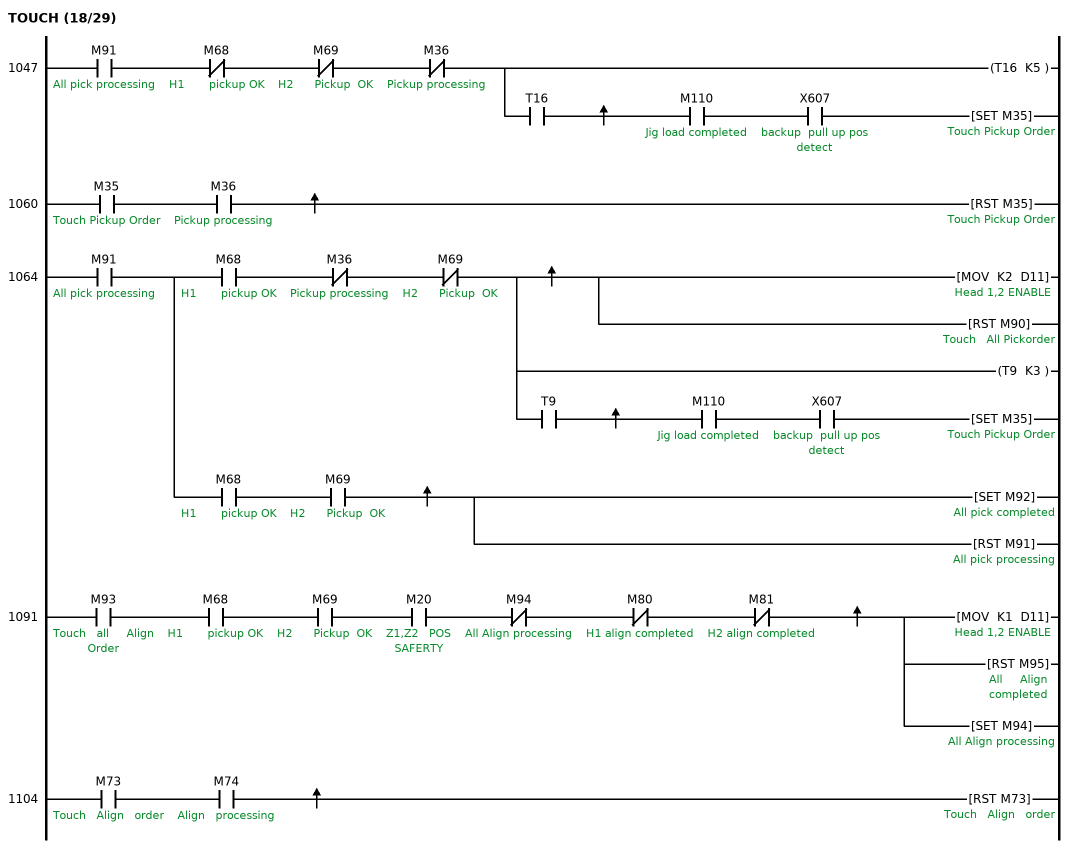
1047  LD      M91  ; All pick processing
      ANI     M68  ; H1       pickup OK
      ANI     M69  ; H2      Pickup  OK
      ANI     M36  ; Pickup processing
      OUT     T16 K5
      AND     T16
      MEP
      AND     M110  ; Jig load completed
      AND     X607  ; backup  pull up pos     detect
      SET     M35  ; Touch Pickup Order
1060  LD      M35  ; Touch Pickup Order
      AND     M36  ; Pickup processing
      MEP
      RST     M35  ; Touch Pickup Order
1064  LD      M91  ; All pick processing
      MPS
      AND     M68  ; H1       pickup OK
      ANI     M36  ; Pickup processing
      ANI     M69  ; H2      Pickup  OK
      MPS
      MEP
      MOV     K2 D11
      RST     M90  ; Touch   All Pickorder
      MPP
      OUT     T9 K3
      AND     T9
      MEP
      AND     M110  ; Jig load completed
      AND     X607  ; backup  pull up pos     detect
      SET     M35  ; Touch Pickup Order
      MPP
      AND     M68  ; H1       pickup OK
      AND     M69  ; H2      Pickup  OK
      MEP
      SET     M92  ; All pick completed
      RST     M91  ; All pick processing
1091  LD      M93  ; Touch   all     Align   Order
      AND     M68  ; H1       pickup OK
      AND     M69  ; H2      Pickup  OK
      AND     M20  ; Z1,Z2   POS     SAFERTY
      ANI     M94  ; All Align processing
      ANI     M80  ; H1 align completed
      ANI     M81  ; H2 align completed
      MEP
      MOV     K1 D11
      RST     M95  ; All     Align   completed
      SET     M94  ; All Align processing
1104  LD      M73  ; Touch   Align   order
      AND     M74  ; Align   processing
      MEP
      RST     M73  ; Touch   Align   order
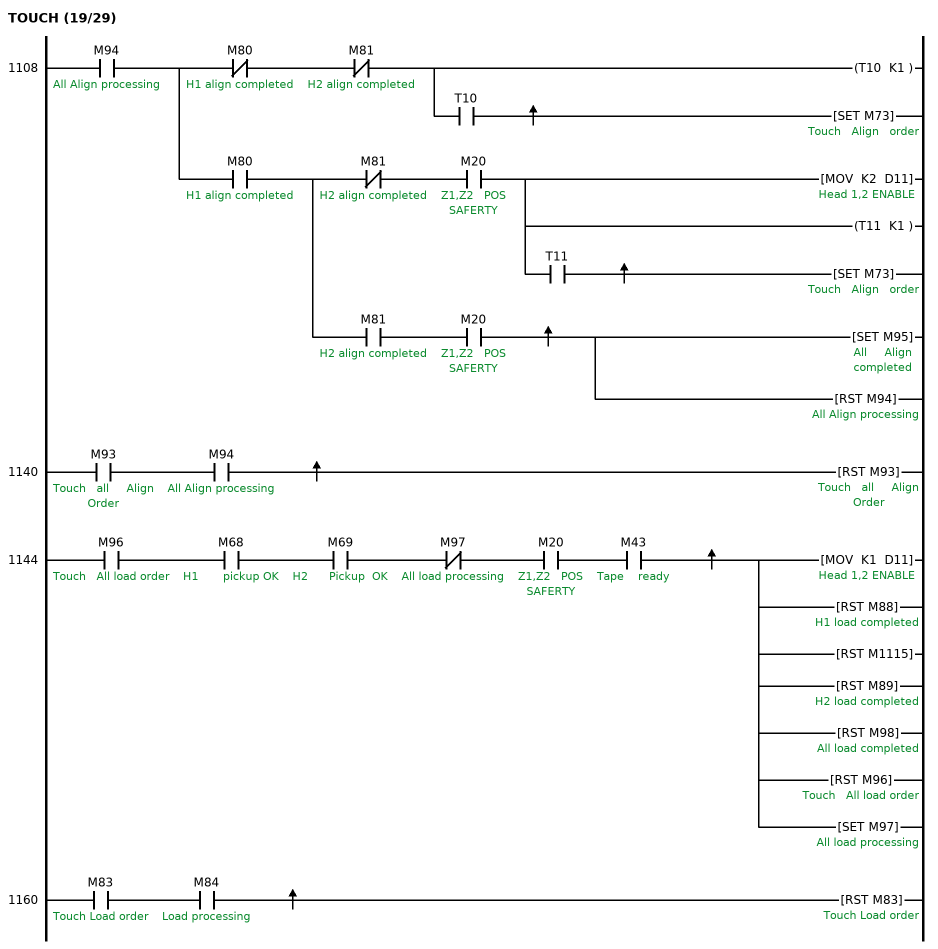
1108  LD      M94  ; All Align processing
      MPS
      ANI     M80  ; H1 align completed
      ANI     M81  ; H2 align completed
      OUT     T10 K1
      AND     T10
      MEP
      SET     M73  ; Touch   Align   order
      MPP
      AND     M80  ; H1 align completed
      MPS
      ANI     M81  ; H2 align completed
      AND     M20  ; Z1,Z2   POS     SAFERTY
      MOV     K2 D11
      OUT     T11 K1
      AND     T11
      MEP
      SET     M73  ; Touch   Align   order
      MPP
      AND     M81  ; H2 align completed
      AND     M20  ; Z1,Z2   POS     SAFERTY
      MEP
      SET     M95  ; All     Align   completed
      RST     M94  ; All Align processing
1140  LD      M93  ; Touch   all     Align   Order
      AND     M94  ; All Align processing
      MEP
      RST     M93  ; Touch   all     Align   Order
1144  LD      M96  ; Touch   All load order
      AND     M68  ; H1       pickup OK
      AND     M69  ; H2      Pickup  OK
      ANI     M97  ; All load processing
      AND     M20  ; Z1,Z2   POS     SAFERTY
      AND     M43  ; Tape    ready
      MEP
      MOV     K1 D11
      RST     M88  ; H1 load completed
      RST     M1115
      RST     M89  ; H2 load completed
      RST     M98  ; All load completed
      RST     M96  ; Touch   All load order
      SET     M97  ; All load processing
1160  LD      M83  ; Touch Load order
      AND     M84  ; Load processing
      MEP
      RST     M83  ; Touch Load order
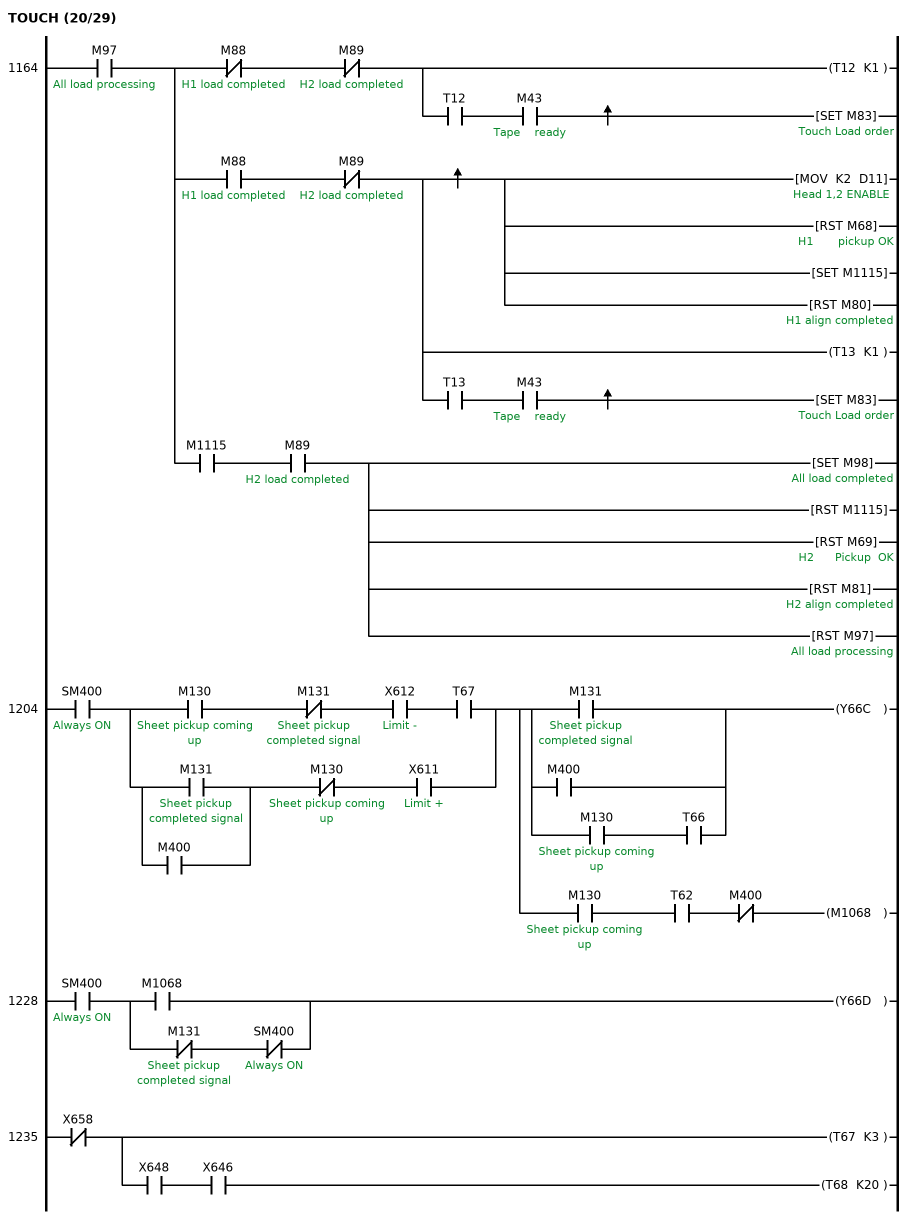
1164  LD      M97  ; All load processing
      MPS
      ANI     M88  ; H1 load completed
      ANI     M89  ; H2 load completed
      OUT     T12 K1
      AND     T12
      AND     M43  ; Tape    ready
      MEP
      SET     M83  ; Touch Load order
      MRD
      AND     M88  ; H1 load completed
      ANI     M89  ; H2 load completed
      MPS
      MEP
      MOV     K2 D11
      RST     M68  ; H1       pickup OK
      SET     M1115
      RST     M80  ; H1 align completed
      MPP
      OUT     T13 K1
      AND     T13
      AND     M43  ; Tape    ready
      MEP
      SET     M83  ; Touch Load order
      MPP
      AND     M1115
      AND     M89  ; H2 load completed
      SET     M98  ; All load completed
      RST     M1115
      RST     M69  ; H2      Pickup  OK
      RST     M81  ; H2 align completed
      RST     M97  ; All load processing
1204  LD      SM400  ; Always ON
      LD      M130  ; Sheet pickup coming up
      ANI     M131  ; Sheet pickup completed signal
      AND     X612  ; Limit -
      AND     T67
      LD      M131  ; Sheet pickup completed signal
      OR      M400
      ANI     M130  ; Sheet pickup coming up
      AND     X611  ; Limit +
      ORB
      ANB
      MPS
      LD      M131  ; Sheet pickup completed signal
      OR      M400
      LD      M130  ; Sheet pickup coming up
      AND     T66
      ORB
      ANB
      OUT     Y66C
      MPP
      AND     M130  ; Sheet pickup coming up
      AND     T62
      ANI     M400
      OUT     M1068
1228  LD      SM400  ; Always ON
      LD      M1068
      LDI     M131  ; Sheet pickup completed signal
      ANI     SM400  ; Always ON
      ORB
      ANB
      OUT     Y66D
1235  LDI     X658
      OUT     T67 K3
      AND     X648
      AND     X646
      OUT     T68 K20
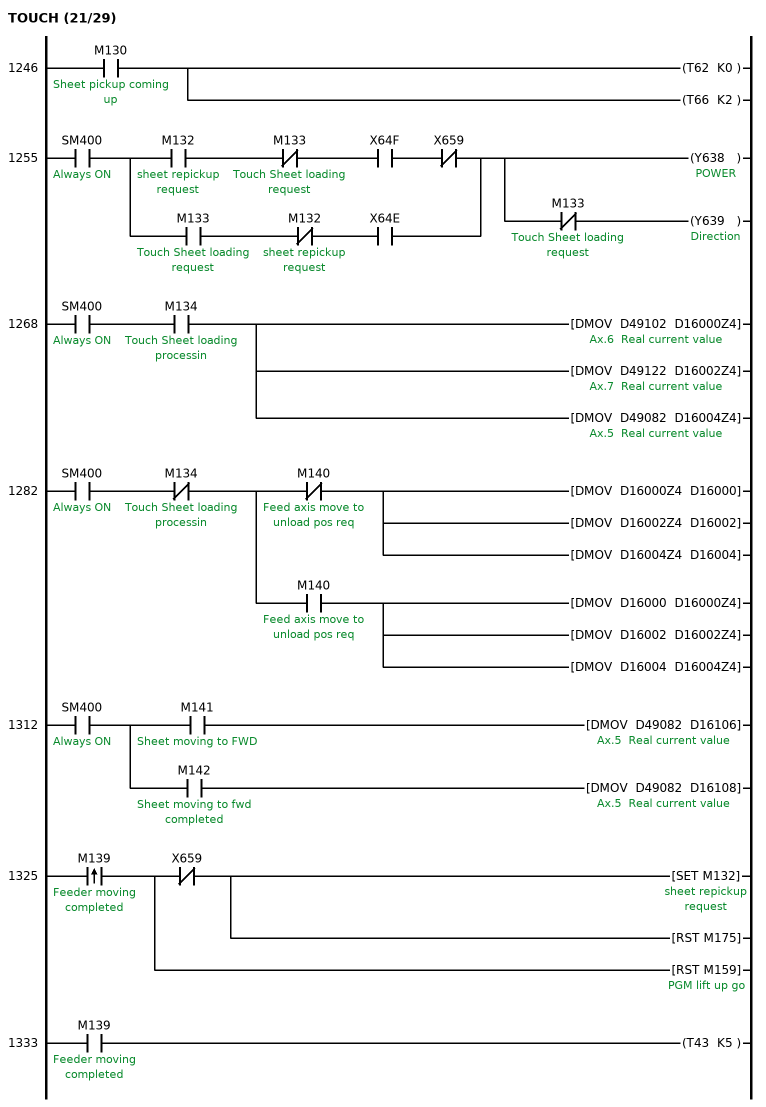
1246  LD      M130  ; Sheet pickup coming up
      OUT     T62 K0
      OUT     T66 K2
1255  LD      SM400  ; Always ON
      LD      M132  ; sheet repickup request
      ANI     M133  ; Touch Sheet loading request
      AND     X64F
      ANI     X659
      LD      M133  ; Touch Sheet loading request
      ANI     M132  ; sheet repickup request
      AND     X64E
      ORB
      ANB
      OUT     Y638  ; POWER
      ANI     M133  ; Touch Sheet loading request
      OUT     Y639  ; Direction
1268  LD      SM400  ; Always ON
      AND     M134  ; Touch Sheet loading processin
      DMOV    D49102 D16000Z4
      DMOV    D49122 D16002Z4
      DMOV    D49082 D16004Z4  ; Ax.5  Real current value
1282  LD      SM400  ; Always ON
      ANI     M134  ; Touch Sheet loading processin
      MPS
      ANI     M140  ; Feed axis move to unload pos req
      DMOV    D16000Z4 D16000
      DMOV    D16002Z4 D16002
      DMOV    D16004Z4 D16004
      MPP
      AND     M140  ; Feed axis move to unload pos req
      DMOV    D16000 D16000Z4
      DMOV    D16002 D16002Z4
      DMOV    D16004 D16004Z4
1312  LD      SM400  ; Always ON
      MPS
      AND     M141  ; Sheet moving to FWD
      DMOV    D49082 D16106
      MPP
      AND     M142  ; Sheet moving to fwd completed
      DMOV    D49082 D16108
1325  LDP     M139  ; Feeder moving completed
      MPS
      ANI     X659
      SET     M132  ; sheet repickup request
      RST     M175
      MPP
      RST     M159  ; PGM lift up go
1333  LD      M139  ; Feeder moving completed
      OUT     T43 K5
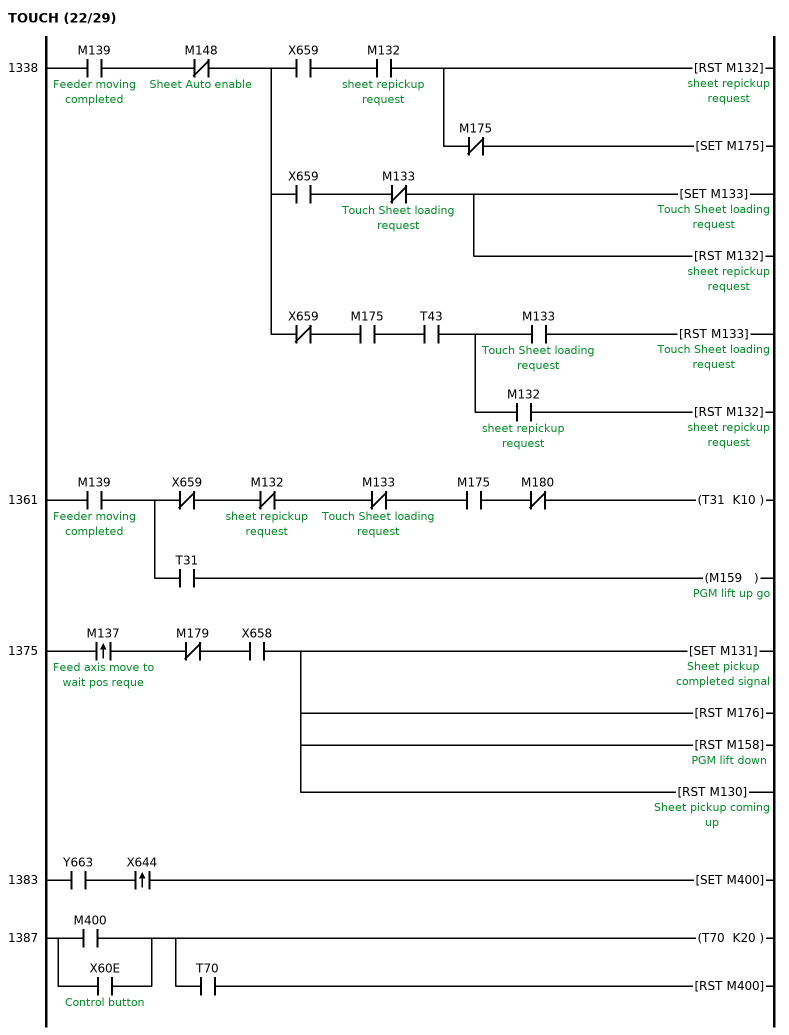
1338  LD      M139  ; Feeder moving completed
      ANI     M148  ; Sheet Auto enable
      MPS
      AND     X659
      AND     M132  ; sheet repickup request
      RST     M132  ; sheet repickup request
      ANI     M175
      SET     M175
      MRD
      AND     X659
      ANI     M133  ; Touch Sheet loading request
      SET     M133  ; Touch Sheet loading request
      RST     M132  ; sheet repickup request
      MPP
      ANI     X659
      AND     M175
      AND     T43
      MPS
      AND     M133  ; Touch Sheet loading request
      RST     M133  ; Touch Sheet loading request
      MPP
      AND     M132  ; sheet repickup request
      RST     M132  ; sheet repickup request
1361  LD      M139  ; Feeder moving completed
      MPS
      ANI     X659
      ANI     M132  ; sheet repickup request
      ANI     M133  ; Touch Sheet loading request
      AND     M175
      ANI     M180
      OUT     T31 K10
      MPP
      AND     T31
      OUT     M159  ; PGM lift up go
1375  LDP     M137  ; Feed axis move to wait pos reque
      ANI     M179
      AND     X658
      SET     M131  ; Sheet pickup completed signal
      RST     M176
      RST     M158  ; PGM lift down
      RST     M130  ; Sheet pickup coming up
1383  LD      Y663
      ANDP    X644
      SET     M400
1387  LD      M400
      OR      X60E  ; Control button
      OUT     T70 K20
      AND     T70
      RST     M400
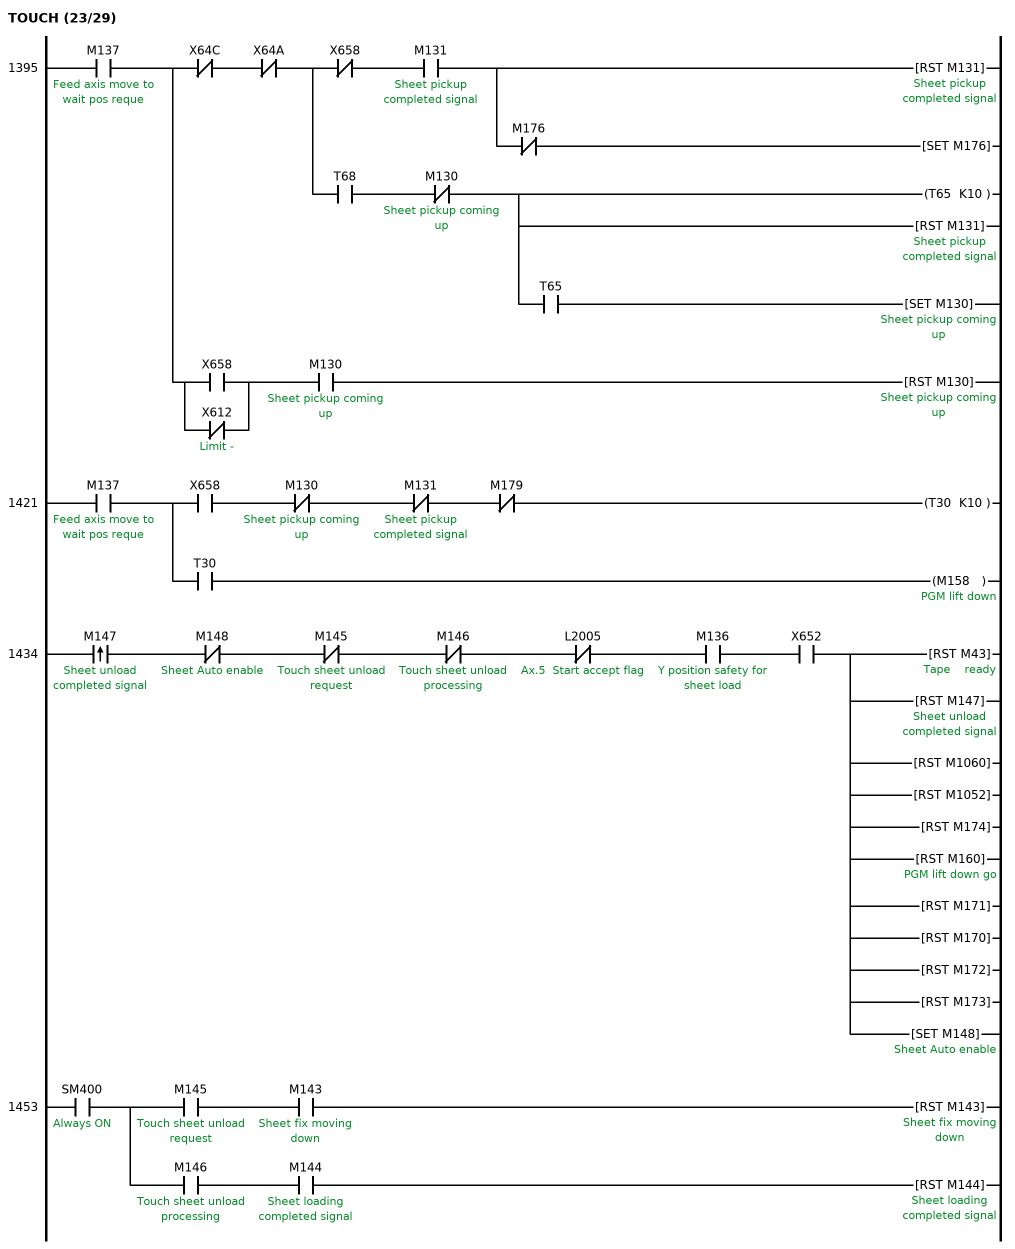
1395  LD      M137  ; Feed axis move to wait pos reque
      MPS
      ANI     X64C
      ANI     X64A
      MPS
      ANI     X658
      AND     M131  ; Sheet pickup completed signal
      RST     M131  ; Sheet pickup completed signal
      ANI     M176
      SET     M176
      MPP
      AND     T68
      ANI     M130  ; Sheet pickup coming up
      OUT     T65 K10
      RST     M131  ; Sheet pickup completed signal
      AND     T65
      SET     M130  ; Sheet pickup coming up
      MPP
      LD      X658
      ORI     X612  ; Limit -
      ANB
      AND     M130  ; Sheet pickup coming up
      RST     M130  ; Sheet pickup coming up
1421  LD      M137  ; Feed axis move to wait pos reque
      MPS
      AND     X658
      ANI     M130  ; Sheet pickup coming up
      ANI     M131  ; Sheet pickup completed signal
      ANI     M179
      OUT     T30 K10
      MPP
      AND     T30
      OUT     M158  ; PGM lift down
1434  LDP     M147  ; Sheet unload completed signal
      ANI     M148  ; Sheet Auto enable
      ANI     M145  ; Touch sheet unload request
      ANI     M146  ; Touch sheet unload processing
      ANI     L2005  ; Ax.5  Start accept flag
      AND     M136  ; Y position safety for sheet load
      AND     X652
      RST     M43  ; Tape    ready
      RST     M147  ; Sheet unload completed signal
      RST     M1060
      RST     M1052
      RST     M174
      RST     M160  ; PGM lift down go
      RST     M171
      RST     M170
      RST     M172
      RST     M173
      SET     M148  ; Sheet Auto enable
1453  LD      SM400  ; Always ON
      MPS
      AND     M145  ; Touch sheet unload request
      AND     M143  ; Sheet fix moving down
      RST     M143  ; Sheet fix moving down
      MPP
      AND     M146  ; Touch sheet unload processing
      AND     M144  ; Sheet loading completed signal
      RST     M144  ; Sheet loading completed signal
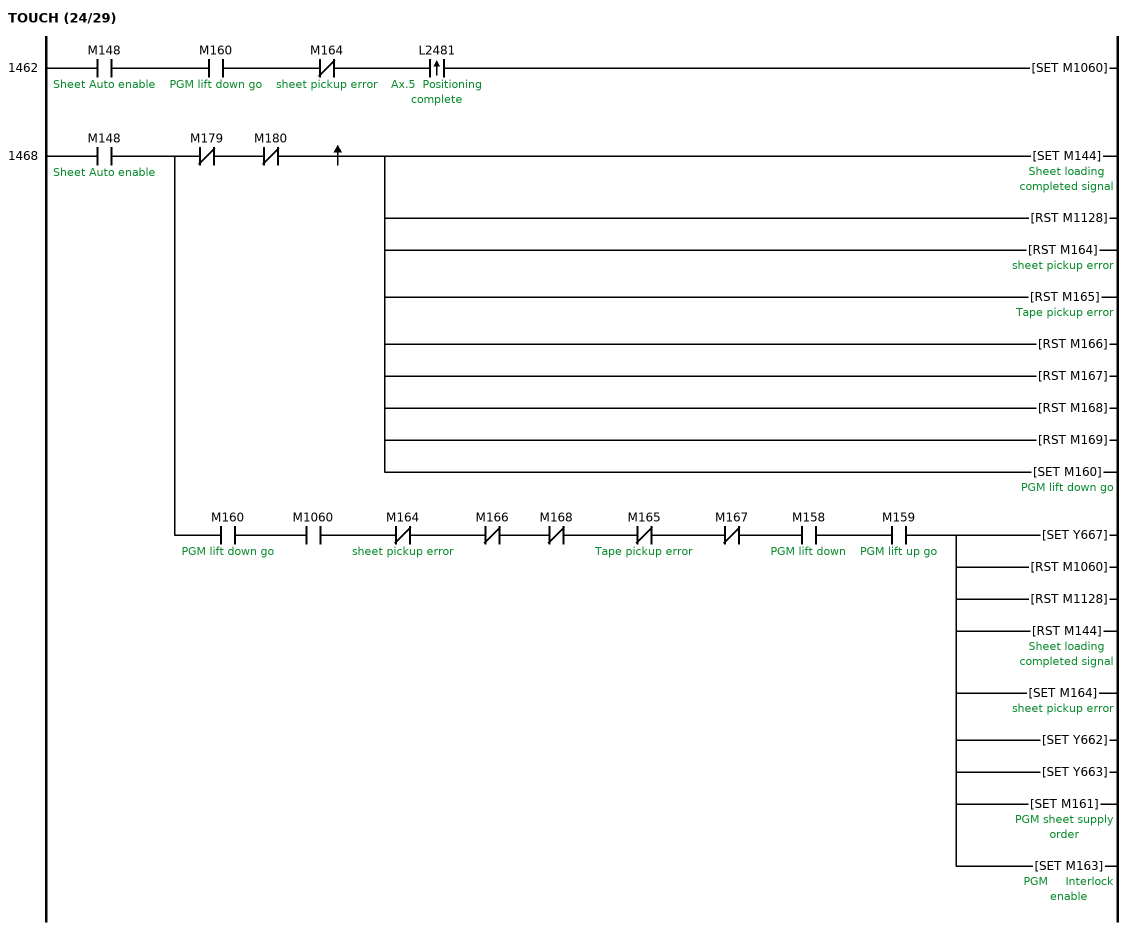
1462  LD      M148  ; Sheet Auto enable
      AND     M160  ; PGM lift down go
      ANI     M164  ; sheet pickup error
      ANDP    L2481  ; Ax.5  Positioning complete
      SET     M1060
1468  LD      M148  ; Sheet Auto enable
      MPS
      ANI     M179
      ANI     M180
      MEP
      SET     M144  ; Sheet loading completed signal
      RST     M1128
      RST     M164  ; sheet pickup error
      RST     M165  ; Tape pickup error
      RST     M166
      RST     M167
      RST     M168
      RST     M169
      SET     M160  ; PGM lift down go
      MPP
      AND     M160  ; PGM lift down go
      AND     M1060
      ANI     M164  ; sheet pickup error
      ANI     M166
      ANI     M168
      ANI     M165  ; Tape pickup error
      ANI     M167
      AND     M158  ; PGM lift down
      AND     M159  ; PGM lift up go
      SET     Y667
      RST     M1060
      RST     M1128
      RST     M144  ; Sheet loading completed signal
      SET     M164  ; sheet pickup error
      SET     Y662
      SET     Y663
      SET     M161  ; PGM sheet supply order
      SET     M163  ; PGM     Interlock enable
